C03648=1141.672,169.284,-60.274,-178.490,7.173,148.902
C03649=1141.677,169.034,-60.251,-178.493,7.171,148.902
C03650=1141.681,168.786,-60.228,-178.496,7.169,148.903
C03651=1141.685,168.537,-60.206,-178.499,7.167,148.903
C03652=1141.690,168.288,-60.185,-178.501,7.165,148.903
C03653=1141.695,168.039,-60.162,-178.505,7.162,148.903
C03654=1141.699,167.790,-60.139,-178.507,7.160,148.904
C03655=1141.704,167.541,-60.118,-178.510,7.158,148.904
C03656=1141.708,167.292,-60.096,-178.513,7.156,148.904
C03657=1141.714,167.043,-60.073,-178.516,7.154,148.905
C03658=1141.718,166.794,-60.051,-178.518,7.151,148.905
C03659=1141.723,166.546,-60.029,-178.521,7.150,148.905
C03660=1141.727,166.296,-60.007,-178.524,7.147,148.906
C03661=1141.733,166.047,-59.985,-178.527,7.145,148.906
C03662=1141.737,165.798,-59.963,-178.529,7.143,148.906
C03663=1141.742,165.549,-59.941,-178.533,7.141,148.906
C03664=1141.746,165.300,-59.919,-178.535,7.139,148.907
C03665=1141.751,165.051,-59.897,-178.538,7.137,148.907
C03666=1141.755,164.802,-59.875,-178.541,7.134,148.907
C03667=1141.761,164.553,-59.853,-178.544,7.133,148.908
C03668=1141.765,164.304,-59.830,-178.547,7.130,148.908
C03669=1141.770,164.056,-59.808,-178.549,7.128,148.908
C03670=1141.774,163.806,-59.786,-178.552,7.126,148.909
C03671=1141.779,163.558,-59.765,-178.555,7.124,148.909
C03672=1141.783,163.308,-59.743,-178.558,7.122,148.909
C03673=1141.788,163.060,-59.721,-178.560,7.120,148.909
C03674=1141.792,162.811,-59.699,-178.563,7.118,148.910
C03675=1141.798,162.562,-59.677,-178.566,7.116,148.910
C03676=1141.803,162.313,-59.655,-178.569,7.113,148.911
C03677=1141.807,162.063,-59.634,-178.572,7.111,148.911
C03678=1141.812,161.814,-59.612,-178.574,7.110,148.911
C03679=1141.816,161.565,-59.590,-178.578,7.107,148.911
C03680=1141.821,161.316,-59.568,-178.580,7.105,148.912
C03681=1141.826,161.067,-59.546,-178.583,7.103,148.912
C03682=1141.830,160.818,-59.524,-178.586,7.101,148.912
C03683=1141.835,160.570,-59.503,-178.589,7.099,148.913
C03684=1141.840,160.320,-59.481,-178.591,7.097,148.913
C03685=1141.844,160.072,-59.459,-178.594,7.094,148.913
C03686=1141.849,159.822,-59.438,-178.597,7.093,148.914
C03687=1141.854,159.573,-59.416,-178.599,7.091,148.914
C03688=1141.859,159.324,-59.394,-178.603,7.088,148.914
C03689=1141.863,159.075,-59.372,-178.605,7.087,148.915
C03690=1141.868,158.827,-59.351,-178.608,7.085,148.915
C03691=1141.873,158.578,-59.329,-178.611,7.082,148.915
C03692=1141.877,158.328,-59.308,-178.614,7.080,148.916
C03693=1141.882,158.079,-59.286,-178.616,7.079,148.916
C03694=1141.887,157.810,-59.263,-178.620,7.076,148.916
C03695=1141.892,157.541,-59.239,-178.623,7.074,148.917
C03696=1141.897,157.272,-59.216,-178.625,7.072,148.917
C03697=1141.902,157.003,-59.193,-178.629,7.069,148.917
C03698=1141.907,156.754,-59.171,-178.631,7.067,148.918
C03699=1141.911,156.505,-59.149,-178.634,7.066,148.918
C03700=1141.916,156.256,-59.129,-178.637,7.063,148.918
C03701=1141.921,156.008,-59.107,-178.640,7.061,148.919
C03702=1141.925,155.758,-59.085,-178.642,7.059,148.919
C03703=1141.930,155.509,-59.064,-178.646,7.057,148.919
C03704=1141.935,155.260,-59.042,-178.648,7.055,148.920
C03705=1141.940,155.012,-59.021,-178.651,7.053,148.920
C03706=1141.945,154.762,-58.999,-178.654,7.051,148.920
C03707=1141.949,154.513,-58.978,-178.656,7.049,148.921
C03708=1141.954,154.264,-58.957,-178.659,7.047,148.921
C03709=1141.959,154.015,-58.936,-178.662,7.045,148.921
C03710=1141.963,153.765,-58.914,-178.665,7.043,148.922
C03711=1141.968,153.517,-58.893,-178.668,7.041,148.922
C03712=1141.973,153.268,-58.872,-178.671,7.039,148.922
C03713=1141.977,153.019,-58.851,-178.673,7.036,148.923
C03714=1141.982,152.769,-58.829,-178.676,7.035,148.923
C03715=1141.987,152.521,-58.808,-178.679,7.033,148.923
C03716=1141.992,152.271,-58.787,-178.682,7.031,148.924
C03717=1141.996,152.023,-58.766,-178.685,7.029,148.924
C03718=1142.001,151.773,-58.744,-178.688,7.027,148.925
C03719=1142.006,151.524,-58.722,-178.690,7.025,148.925
C03720=1142.011,151.275,-58.702,-178.693,7.022,148.925
C03721=1142.015,151.027,-58.680,-178.696,7.021,148.925
C03722=1142.020,150.778,-58.659,-178.699,7.019,148.926
C03723=1142.025,150.528,-58.638,-178.701,7.017,148.926
C03724=1142.029,150.279,-58.617,-178.705,7.015,148.927
C03725=1142.034,150.030,-58.596,-178.707,7.013,148.927
C03726=1142.039,149.781,-58.574,-178.709,7.011,148.927
C03727=1142.043,149.532,-58.554,-178.712,7.009,148.927
C03728=1142.048,149.282,-58.533,-178.716,7.007,148.928
C03729=1142.053,149.034,-58.511,-178.718,7.005,148.928
C03730=1142.057,148.785,-58.491,-178.721,7.003,148.929
C03731=1142.062,148.536,-58.470,-178.724,7.002,148.929
C03732=1142.068,148.286,-58.449,-178.727,6.999,148.929
C03733=1142.072,148.038,-58.428,-178.729,6.997,148.930
C03734=1142.077,147.789,-58.407,-178.732,6.995,148.930
C03735=1142.081,147.539,-58.385,-178.735,6.994,148.930
C03736=1142.086,147.290,-58.365,-178.738,6.991,148.931
C03737=1142.091,147.041,-58.343,-178.741,6.989,148.931
C03738=1142.095,146.792,-58.323,-178.743,6.988,148.931
C03739=1142.100,146.543,-58.302,-178.746,6.986,148.932
C03740=1142.105,146.294,-58.282,-178.749,6.983,148.932
C03741=1142.110,146.045,-58.261,-178.752,6.981,148.932
C03742=1142.115,145.796,-58.239,-178.754,6.980,148.933
C03743=1142.119,145.547,-58.219,-178.757,6.978,148.933
C03744=1142.124,145.297,-58.197,-178.760,6.975,148.934
C03745=1142.128,145.048,-58.177,-178.763,6.974,148.934
C03746=1142.133,144.799,-58.156,-178.766,6.972,148.934
C03747=1142.138,144.550,-58.135,-178.768,6.970,148.935
C03748=1142.143,144.301,-58.115,-178.771,6.969,148.935
C03749=1142.147,144.053,-58.093,-178.774,6.966,148.935
C03750=1142.152,143.803,-58.072,-178.777,6.964,148.936
C03751=1142.157,143.554,-58.052,-178.779,6.962,148.936
C03752=1142.162,143.305,-58.031,-178.782,6.961,148.936
C03753=1142.166,143.056,-58.011,-178.785,6.958,148.937
C03754=1142.172,142.807,-57.990,-178.788,6.956,148.937
C03755=1142.176,142.558,-57.969,-178.791,6.955,148.938
C03756=1142.180,142.309,-57.949,-178.794,6.953,148.938
C03757=1142.186,142.060,-57.928,-178.796,6.951,148.938
C03758=1142.190,141.811,-57.908,-178.800,6.949,148.939
C03759=1142.195,141.562,-57.887,-178.802,6.947,148.939
C03760=1142.200,141.313,-57.866,-178.805,6.945,148.939
C03761=1142.204,141.064,-57.846,-178.807,6.943,148.940
C03762=1142.209,140.814,-57.825,-178.810,6.942,148.940
C03763=1142.214,140.565,-57.805,-178.813,6.939,148.940
C03764=1142.219,140.316,-57.784,-178.816,6.937,148.941
C03765=1142.224,140.067,-57.764,-178.819,6.936,148.941
C03766=1142.228,139.818,-57.744,-178.821,6.934,148.942
C03767=1142.233,139.568,-57.723,-178.824,6.932,148.942
C03768=1142.238,139.319,-57.702,-178.827,6.931,148.942
C03769=1142.242,139.070,-57.682,-178.830,6.928,148.943
C03770=1142.247,138.821,-57.661,-178.833,6.926,148.943
C03771=1142.252,138.572,-57.641,-178.836,6.925,148.944
C03772=1142.256,138.323,-57.621,-178.838,6.923,148.944
C03773=1142.262,138.073,-57.600,-178.841,6.921,148.944
C03774=1142.266,137.824,-57.580,-178.843,6.919,148.944
C03775=1142.271,137.576,-57.559,-178.847,6.917,148.945
C03776=1142.275,137.327,-57.539,-178.849,6.915,148.945
C03777=1142.280,137.077,-57.519,-178.852,6.913,148.946
C03778=1142.285,136.828,-57.498,-178.855,6.912,148.946
C03779=1142.289,136.579,-57.478,-178.857,6.910,148.946
C03780=1142.294,136.330,-57.457,-178.860,6.908,148.947
C03781=1142.300,136.081,-57.438,-178.864,6.906,148.947
C03782=1142.304,135.832,-57.417,-178.866,6.904,148.948
C03783=1142.309,135.583,-57.397,-178.869,6.902,148.948
C03784=1142.313,135.333,-57.377,-178.872,6.901,148.948
C03785=1142.319,135.084,-57.356,-178.874,6.899,148.949
C03786=1142.323,134.835,-57.336,-178.877,6.897,148.949
C03787=1142.328,134.585,-57.316,-178.880,6.895,148.950
C03788=1142.332,134.336,-57.296,-178.883,6.893,148.950
C03789=1142.337,134.088,-57.275,-178.886,6.891,148.950
C03790=1142.343,133.838,-57.256,-178.889,6.890,148.951
C03791=1142.347,133.589,-57.235,-178.891,6.888,148.951
C03792=1142.352,133.340,-57.215,-178.894,6.886,148.951
C03793=1142.356,133.091,-57.195,-178.897,6.884,148.952
C03794=1142.361,132.842,-57.175,-178.899,6.883,148.952
C03795=1142.366,132.592,-57.155,-178.903,6.880,148.953
C03796=1142.371,132.344,-57.135,-178.905,6.878,148.953
C03797=1142.376,132.094,-57.115,-178.908,6.876,148.953
C03798=1142.381,131.826,-57.093,-178.911,6.875,148.954
C03799=1142.386,131.557,-57.071,-178.914,6.873,148.954
C03800=1142.391,131.289,-57.050,-178.917,6.871,148.955
C03801=1142.396,131.021,-57.029,-178.920,6.869,148.955
C03802=1142.401,130.771,-57.008,-178.922,6.867,148.955
C03803=1142.406,130.522,-56.988,-178.926,6.865,148.956
C03804=1142.411,130.273,-56.969,-178.928,6.863,148.956
C03805=1142.416,130.023,-56.949,-178.931,6.862,148.957
C03806=1142.420,129.774,-56.929,-178.934,6.860,148.957
C03807=1142.425,129.525,-56.909,-178.937,6.858,148.957
C03808=1142.429,129.276,-56.889,-178.939,6.856,148.958
C03809=1142.435,129.027,-56.869,-178.942,6.855,148.958
C03810=1142.439,128.778,-56.849,-178.945,6.853,148.959
C03811=1142.444,128.528,-56.829,-178.947,6.851,148.959
C03812=1142.449,128.279,-56.810,-178.950,6.850,148.959
C03813=1142.454,128.031,-56.790,-178.953,6.847,148.960
C03814=1142.459,127.781,-56.770,-178.956,6.845,148.960
C03815=1142.463,127.532,-56.750,-178.959,6.844,148.961
C03816=1142.468,127.283,-56.730,-178.962,6.842,148.961
C03817=1142.473,127.034,-56.711,-178.964,6.840,148.961
C03818=1142.478,126.784,-56.691,-178.967,6.839,148.962
C03819=1142.483,126.535,-56.671,-178.970,6.837,148.962
C03820=1142.488,126.286,-56.651,-178.973,6.835,148.963
C03821=1142.492,126.037,-56.632,-178.975,6.834,148.963
C03822=1142.497,125.787,-56.612,-178.978,6.832,148.963
C03823=1142.501,125.539,-56.592,-178.981,6.830,148.964
C03824=1142.506,125.290,-56.573,-178.983,6.829,148.964
C03825=1142.511,125.040,-56.553,-178.986,6.827,148.965
C03826=1142.516,124.791,-56.534,-178.989,6.824,148.965
C03827=1142.521,124.542,-56.514,-178.992,6.823,148.965
C03828=1142.525,124.293,-56.494,-178.995,6.821,148.966
C03829=1142.530,124.043,-56.474,-178.998,6.819,148.966
C03830=1142.535,123.794,-56.455,-179.000,6.818,148.967
C03831=1142.539,123.545,-56.436,-179.003,6.816,148.967
C03832=1142.544,123.295,-56.416,-179.006,6.814,148.967
C03833=1142.550,123.047,-56.397,-179.009,6.812,148.968
C03834=1142.554,122.797,-56.377,-179.011,6.811,148.968
C03835=1142.559,122.549,-56.357,-179.014,6.809,148.969
C03836=1142.564,122.299,-56.338,-179.017,6.807,148.969
C03837=1142.568,122.050,-56.319,-179.020,6.806,148.970
C03838=1142.573,121.801,-56.299,-179.023,6.804,148.970
C03839=1142.578,121.552,-56.280,-179.025,6.803,148.970
C03840=1142.583,121.302,-56.260,-179.028,6.801,148.971
C03841=1142.588,121.053,-56.241,-179.031,6.799,148.971
C03842=1142.592,120.804,-56.222,-179.034,6.798,148.972
C03843=1142.598,120.555,-56.202,-179.036,6.796,148.972
C03844=1142.602,120.305,-56.183,-179.039,6.794,148.972
C03845=1142.607,120.056,-56.163,-179.042,6.792,148.973
C03846=1142.612,119.807,-56.144,-179.045,6.790,148.973
C03847=1142.616,119.558,-56.125,-179.048,6.788,148.974
C03848=1142.622,119.309,-56.105,-179.050,6.787,148.974
C03849=1142.627,119.059,-56.086,-179.053,6.785,148.974
C03850=1142.631,118.811,-56.067,-179.056,6.783,148.975
C03851=1142.636,118.561,-56.047,-179.059,6.782,148.975
C03852=1142.641,118.312,-56.028,-179.061,6.780,148.976
C03853=1142.645,118.063,-56.009,-179.064,6.778,148.976
C03854=1142.650,117.813,-55.990,-179.067,6.776,148.976
C03855=1142.656,117.564,-55.971,-179.070,6.775,148.977
C03856=1142.660,117.315,-55.952,-179.073,6.773,148.977
C03857=1142.665,117.066,-55.932,-179.075,6.772,148.978
C03858=1142.670,116.816,-55.913,-179.078,6.770,148.978
C03859=1142.674,116.568,-55.894,-179.081,6.768,148.979
C03860=1142.679,116.318,-55.874,-179.084,6.767,148.979
C03861=1142.685,116.069,-55.856,-179.086,6.765,148.979
C03862=1142.689,115.819,-55.837,-179.089,6.763,148.980
C03863=1142.694,115.571,-55.818,-179.092,6.762,148.980
C03864=1142.699,115.321,-55.798,-179.095,6.760,148.981
C03865=1142.703,115.072,-55.779,-179.097,6.758,148.981
C03866=1142.708,114.822,-55.760,-179.100,6.757,148.981
C03867=1142.713,114.574,-55.742,-179.103,6.755,148.982
C03868=1142.718,114.324,-55.722,-179.106,6.754,148.983
C03869=1142.723,114.075,-55.704,-179.109,6.752,148.983
C03870=1142.727,113.825,-55.684,-179.111,6.750,148.983
C03871=1142.733,113.576,-55.665,-179.114,6.748,148.984
C03872=1142.737,113.328,-55.646,-179.117,6.747,148.984
C03873=1142.742,113.078,-55.627,-179.120,6.745,148.985
C03874=1142.747,112.829,-55.609,-179.122,6.743,148.985
C03875=1142.752,112.580,-55.589,-179.125,6.742,148.985
C03876=1142.757,112.330,-55.571,-179.127,6.741,148.986
C03877=1142.761,112.081,-55.551,-179.130,6.739,148.986
C03878=1142.766,111.832,-55.533,-179.133,6.738,148.987
C03879=1142.772,111.583,-55.514,-179.136,6.736,148.987
C03880=1142.776,111.334,-55.495,-179.139,6.734,148.988
C03881=1142.781,111.084,-55.476,-179.141,6.733,148.988
C03882=1142.785,110.835,-55.457,-179.144,6.731,148.988
C03883=1142.791,110.585,-55.439,-179.147,6.729,148.989
C03884=1142.796,110.337,-55.420,-179.149,6.728,148.989
C03885=1142.800,110.087,-55.400,-179.152,6.726,148.990
C03886=1142.805,109.838,-55.382,-179.155,6.724,148.990
C03887=1142.810,109.588,-55.363,-179.158,6.723,148.991
C03888=1142.815,109.339,-55.345,-179.161,6.721,148.991
C03889=1142.820,109.091,-55.326,-179.164,6.720,148.992
C03890=1142.825,108.841,-55.307,-179.166,6.718,148.992
C03891=1142.829,108.592,-55.289,-179.169,6.716,148.992
C03892=1142.835,108.342,-55.270,-179.172,6.715,148.993
C03893=1142.839,108.093,-55.251,-179.175,6.713,148.993
C03894=1142.844,107.844,-55.233,-179.177,6.711,148.994
C03895=1142.849,107.595,-55.214,-179.180,6.710,148.994
C03896=1142.853,107.345,-55.195,-179.183,6.708,148.995
C03897=1142.858,107.096,-55.177,-179.185,6.707,148.995
C03898=1142.864,106.847,-55.158,-179.188,6.706,148.995
C03899=1142.868,106.597,-55.140,-179.191,6.704,148.996
C03900=1142.873,106.349,-55.121,-179.194,6.702,148.996
C03901=1142.878,106.099,-55.102,-179.196,6.701,148.997
C03902=1142.883,105.830,-55.083,-179.199,6.699,148.997
C03903=1142.888,105.562,-55.062,-179.202,6.698,148.998
C03904=1142.893,105.294,-55.042,-179.206,6.695,148.998
C03905=1142.899,105.026,-55.022,-179.208,6.693,148.999
C03906=1142.903,104.776,-55.004,-179.211,6.692,148.999
C03907=1142.908,104.527,-54.985,-179.214,6.690,149.000
C03908=1142.914,104.278,-54.967,-179.216,6.690,149.000
C03909=1142.919,104.029,-54.949,-179.219,6.688,149.000
C03910=1142.923,103.779,-54.931,-179.222,6.686,149.001
C03911=1142.928,103.530,-54.912,-179.225,6.684,149.001
C03912=1142.933,103.281,-54.893,-179.227,6.683,149.002
C03913=1142.938,103.031,-54.875,-179.230,6.681,149.002
C03914=1142.942,102.782,-54.857,-179.233,6.680,149.003
C03915=1142.947,102.533,-54.838,-179.236,6.678,149.003
C03916=1142.952,102.284,-54.820,-179.239,6.676,149.004
C03917=1142.958,102.034,-54.802,-179.241,6.675,149.004
C03918=1142.962,101.784,-54.783,-179.244,6.674,149.004
C03919=1142.967,101.536,-54.765,-179.247,6.673,149.005
C03920=1142.971,101.287,-54.747,-179.249,6.671,149.005
C03921=1142.976,101.038,-54.729,-179.252,6.669,149.006
C03922=1142.982,100.788,-54.710,-179.255,6.668,149.006
C03923=1142.986,100.538,-54.692,-179.258,6.666,149.007
C03924=1142.991,100.289,-54.674,-179.260,6.664,149.007
C03925=1142.996,100.040,-54.656,-179.264,6.663,149.008
C03926=1143.001,99.791,-54.638,-179.266,6.661,149.008
C03927=1143.006,99.542,-54.619,-179.268,6.660,149.009
C03928=1143.011,99.292,-54.600,-179.271,6.659,149.009
C03929=1143.016,99.043,-54.582,-179.274,6.657,149.009
C03930=1143.021,98.794,-54.564,-179.277,6.655,149.010
C03931=1143.025,98.544,-54.546,-179.280,6.654,149.010
C03932=1143.030,98.295,-54.528,-179.283,6.652,149.011
C03933=1143.035,98.046,-54.510,-179.285,6.651,149.011
C03934=1143.040,97.796,-54.492,-179.288,6.650,149.012
C03935=1143.044,97.547,-54.474,-179.290,6.648,149.012
C03936=1143.049,97.298,-54.456,-179.293,6.646,149.013
C03937=1143.054,97.049,-54.438,-179.296,6.645,149.013
C03938=1143.059,96.799,-54.420,-179.299,6.643,149.014
C03939=1143.064,96.550,-54.402,-179.302,6.642,149.014
C03940=1143.070,96.301,-54.383,-179.304,6.640,149.014
C03941=1143.074,96.051,-54.365,-179.307,6.639,149.015
C03942=1143.079,95.802,-54.347,-179.310,6.638,149.015
C03943=1143.084,95.553,-54.329,-179.312,6.636,149.016
C03944=1143.089,95.303,-54.311,-179.315,6.635,149.016
C03945=1143.094,95.054,-54.294,-179.318,6.633,149.017
C03946=1143.099,94.804,-54.276,-179.321,6.631,149.017
C03947=1143.104,94.555,-54.258,-179.323,6.629,149.018
C03948=1143.109,94.306,-54.240,-179.326,6.629,149.018
C03949=1143.114,94.057,-54.222,-179.329,6.627,149.019
C03950=1143.119,93.808,-54.204,-179.332,6.626,149.019
C03951=1143.124,93.559,-54.186,-179.334,6.624,149.019
C03952=1143.128,93.309,-54.169,-179.337,6.622,149.020
C03953=1143.132,93.059,-54.151,-179.340,6.622,149.021
C03954=1143.137,92.810,-54.133,-179.342,6.620,149.021
C03955=1143.142,92.561,-54.115,-179.345,6.618,149.021
C03956=1143.147,92.312,-54.097,-179.348,6.617,149.022
C03957=1143.152,92.062,-54.080,-179.351,6.615,149.022
C03958=1143.157,91.813,-54.062,-179.354,6.614,149.023
C03959=1143.162,91.564,-54.044,-179.356,6.613,149.023
C03960=1143.167,91.314,-54.026,-179.359,6.611,149.024
C03961=1143.172,91.065,-54.009,-179.361,6.610,149.024
C03962=1143.177,90.815,-53.991,-179.364,6.608,149.025
C03963=1143.181,90.567,-53.973,-179.367,6.607,149.025
C03964=1143.186,90.317,-53.955,-179.370,6.606,149.026
C03965=1143.191,90.068,-53.938,-179.372,6.604,149.026
C03966=1143.196,89.818,-53.920,-179.375,6.602,149.026
C03967=1143.201,89.569,-53.902,-179.378,6.601,149.027
C03968=1143.206,89.319,-53.885,-179.381,6.599,149.028
C03969=1143.211,89.070,-53.867,-179.383,6.599,149.028
C03970=1143.216,88.821,-53.849,-179.386,6.597,149.028
C03971=1143.221,88.572,-53.832,-179.389,6.595,149.029
C03972=1143.226,88.322,-53.814,-179.392,6.594,149.029
C03973=1143.231,88.073,-53.797,-179.395,6.592,149.030
C03974=1143.236,87.823,-53.779,-179.397,6.591,149.030
C03975=1143.240,87.575,-53.762,-179.399,6.590,149.031
C03976=1143.245,87.325,-53.744,-179.403,6.588,149.031
C03977=1143.250,87.076,-53.726,-179.405,6.587,149.032
C03978=1143.255,86.826,-53.709,-179.408,6.585,149.032
C03979=1143.260,86.578,-53.692,-179.410,6.584,149.033
C03980=1143.265,86.328,-53.675,-179.413,6.582,149.033
C03981=1143.270,86.079,-53.657,-179.416,6.581,149.034
C03982=1143.275,85.829,-53.639,-179.419,6.580,149.034
C03983=1143.280,85.580,-53.622,-179.421,6.579,149.035
C03984=1143.285,85.330,-53.605,-179.424,6.577,149.035
C03985=1143.290,85.081,-53.587,-179.427,6.576,149.036
C03986=1143.295,84.831,-53.570,-179.430,6.574,149.036
C03987=1143.299,84.582,-53.552,-179.432,6.573,149.036
C03988=1143.304,84.333,-53.535,-179.435,6.571,149.037
C03989=1143.309,84.083,-53.517,-179.438,6.570,149.038
C03990=1143.314,83.834,-53.500,-179.441,6.569,149.038
C03991=1143.319,83.585,-53.483,-179.443,6.568,149.038
C03992=1143.324,83.336,-53.465,-179.446,6.566,149.039
C03993=1143.329,83.086,-53.449,-179.449,6.565,149.039
C03994=1143.334,82.837,-53.431,-179.451,6.563,149.040
C03995=1143.339,82.587,-53.414,-179.454,6.562,149.040
C03996=1143.343,82.338,-53.396,-179.456,6.560,149.041
C03997=1143.348,82.089,-53.379,-179.460,6.559,149.041
C03998=1143.354,81.839,-53.362,-179.462,6.558,149.042
C03999=1143.358,81.591,-53.345,-179.464,6.557,149.042
C04000=1143.364,81.341,-53.327,-179.467,6.555,149.043
C04001=1143.368,81.091,-53.311,-179.470,6.554,149.043
C04002=1143.373,80.842,-53.293,-179.473,6.552,149.044
C04003=1143.378,80.592,-53.275,-179.475,6.551,149.044
C04004=1143.383,80.344,-53.259,-179.478,6.549,149.045
C04005=1143.389,80.094,-53.242,-179.481,6.548,149.045
C04006=1143.393,79.826,-53.223,-179.484,6.547,149.046
C04007=1143.398,79.557,-53.204,-179.487,6.545,149.046
C04008=1143.404,79.289,-53.186,-179.490,6.544,149.047
C04009=1143.409,79.020,-53.168,-179.493,6.542,149.047
C04010=1143.414,78.770,-53.151,-179.495,6.541,149.048
C04011=1143.419,78.522,-53.134,-179.498,6.540,149.048
C04012=1143.424,78.272,-53.116,-179.501,6.538,149.049
C04013=1143.429,78.023,-53.100,-179.503,6.537,149.049
C04014=1143.434,77.773,-53.082,-179.506,6.536,149.050
C04015=1143.439,77.524,-53.066,-179.509,6.534,149.050
C04016=1143.444,77.275,-53.049,-179.512,6.533,149.051
C04017=1143.449,77.025,-53.032,-179.514,6.532,149.051
C04018=1143.454,76.776,-53.014,-179.517,6.530,149.052
C04019=1143.459,76.527,-52.998,-179.520,6.529,149.052
C04020=1143.464,76.277,-52.981,-179.522,6.528,149.053
C04021=1143.468,76.028,-52.964,-179.525,6.526,149.053
C04022=1143.474,75.778,-52.947,-179.528,6.525,149.054
C04023=1143.479,75.529,-52.930,-179.530,6.524,149.054
C04024=1143.484,75.279,-52.913,-179.533,6.522,149.055
C04025=1143.488,75.030,-52.896,-179.536,6.521,149.055
C04026=1143.493,74.781,-52.880,-179.539,6.520,149.056
C04027=1143.499,74.531,-52.863,-179.541,6.519,149.056
C04028=1143.503,74.282,-52.846,-179.544,6.517,149.056
C04029=1143.508,74.032,-52.829,-179.547,6.516,149.057
C04030=1143.513,73.783,-52.813,-179.549,6.515,149.058
C04031=1143.518,73.534,-52.796,-179.552,6.513,149.058
C04032=1143.523,73.284,-52.779,-179.555,6.512,149.059
C04033=1143.528,73.035,-52.762,-179.557,6.511,149.059
C04034=1143.533,72.785,-52.745,-179.560,6.509,149.060
C04035=1143.538,72.536,-52.728,-179.563,6.508,149.060
C04036=1143.543,72.287,-52.712,-179.565,6.507,149.061
C04037=1143.548,72.037,-52.695,-179.568,6.506,149.061
C04038=1143.553,71.788,-52.678,-179.571,6.504,149.061
C04039=1143.558,71.539,-52.662,-179.573,6.503,149.062
C04040=1143.563,71.289,-52.645,-179.576,6.502,149.063
C04041=1143.567,71.040,-52.628,-179.579,6.500,149.063
C04042=1143.573,70.791,-52.612,-179.581,6.499,149.063
C04043=1143.577,70.542,-52.595,-179.584,6.498,149.064
C04044=1143.582,70.292,-52.578,-179.587,6.496,149.065
C04045=1143.588,70.042,-52.562,-179.589,6.495,149.065
C04046=1143.592,69.793,-52.546,-179.592,6.494,149.066
C04047=1143.597,69.543,-52.528,-179.595,6.492,149.066
C04048=1143.602,69.294,-52.512,-179.597,6.492,149.066
C04049=1143.607,69.045,-52.495,-179.600,6.490,149.067
C04050=1143.612,68.796,-52.479,-179.603,6.489,149.068
C04051=1143.618,68.546,-52.462,-179.605,6.488,149.068
C04052=1143.622,68.296,-52.446,-179.608,6.486,149.068
C04053=1143.627,68.047,-52.429,-179.611,6.485,149.069
C04054=1143.632,67.798,-52.413,-179.614,6.484,149.070
C04055=1143.637,67.549,-52.396,-179.616,6.482,149.070
C04056=1143.642,67.299,-52.380,-179.619,6.482,149.071
C04057=1143.647,67.049,-52.363,-179.622,6.480,149.071
C04058=1143.652,66.800,-52.347,-179.624,6.479,149.071
C04059=1143.656,66.551,-52.330,-179.627,6.478,149.072
C04060=1143.662,66.301,-52.314,-179.630,6.476,149.073
C04061=1143.667,66.052,-52.297,-179.633,6.475,149.073
C04062=1143.672,65.803,-52.281,-179.635,6.474,149.073
C04063=1143.677,65.553,-52.265,-179.638,6.473,149.074
C04064=1143.682,65.304,-52.249,-179.640,6.472,149.075
C04065=1143.686,65.055,-52.232,-179.643,6.470,149.075
C04066=1143.691,64.805,-52.216,-179.646,6.469,149.076
C04067=1143.697,64.555,-52.199,-179.648,6.468,149.076
C04068=1143.701,64.306,-52.183,-179.651,6.466,149.077
C04069=1143.707,64.057,-52.167,-179.654,6.465,149.077
C04070=1143.711,63.807,-52.150,-179.656,6.464,149.078
C04071=1143.716,63.558,-52.134,-179.659,6.463,149.078
C04072=1143.721,63.308,-52.118,-179.662,6.462,149.079
C04073=1143.726,63.059,-52.102,-179.665,6.460,149.079
C04074=1143.731,62.809,-52.086,-179.667,6.459,149.080
C04075=1143.736,62.561,-52.070,-179.670,6.458,149.080
C04076=1143.742,62.310,-52.053,-179.673,6.457,149.081
C04077=1143.747,62.061,-52.037,-179.675,6.456,149.081
C04078=1143.751,61.811,-52.021,-179.678,6.454,149.082
C04079=1143.756,61.562,-52.005,-179.681,6.453,149.082
C04080=1143.761,61.313,-51.988,-179.683,6.452,149.083
C04081=1143.766,61.064,-51.972,-179.686,6.450,149.083
C04082=1143.771,60.814,-51.956,-179.688,6.450,149.084
C04083=1143.776,60.565,-51.940,-179.691,6.448,149.084
C04084=1143.782,60.315,-51.924,-179.694,6.447,149.085
C04085=1143.786,60.066,-51.908,-179.696,6.446,149.085
C04086=1143.791,59.816,-51.892,-179.699,6.444,149.086
C04087=1143.796,59.567,-51.875,-179.701,6.444,149.086
C04088=1143.801,59.317,-51.860,-179.705,6.442,149.087
C04089=1143.806,59.068,-51.843,-179.707,6.441,149.087
C04090=1143.811,58.819,-51.828,-179.710,6.440,149.088
C04091=1143.816,58.569,-51.811,-179.713,6.439,149.088
C04092=1143.821,58.320,-51.795,-179.715,6.438,149.089
C04093=1143.826,58.070,-51.780,-179.718,6.436,149.089
C04094=1143.831,57.821,-51.763,-179.720,6.436,149.090
C04095=1143.836,57.571,-51.748,-179.723,6.434,149.090
C04096=1143.841,57.321,-51.732,-179.725,6.433,149.091
C04097=1143.846,57.073,-51.715,-179.728,6.432,149.091
C04098=1143.851,56.823,-51.700,-179.731,6.430,149.092
C04099=1143.856,56.573,-51.684,-179.733,6.429,149.092
C04100=1143.861,56.325,-51.668,-179.737,6.428,149.093
C04101=1143.866,56.075,-51.652,-179.739,6.427,149.093
C04102=1143.871,55.825,-51.636,-179.742,6.426,149.094
C04103=1143.876,55.576,-51.620,-179.744,6.425,149.095
C04104=1143.881,55.326,-51.604,-179.747,6.423,149.095
C04105=1143.886,55.077,-51.589,-179.749,6.423,149.095
C04106=1143.891,54.827,-51.573,-179.752,6.421,149.096
C04107=1143.896,54.578,-51.556,-179.754,6.420,149.097
C04108=1143.901,54.329,-51.541,-179.757,6.419,149.097
C04109=1143.906,54.079,-51.526,-179.760,6.418,149.098
C04110=1143.912,53.811,-51.509,-179.763,6.417,149.098
C04111=1143.917,53.542,-51.491,-179.766,6.415,149.099
C04112=1143.922,53.273,-51.474,-179.769,6.414,149.099
C04113=1143.928,53.005,-51.457,-179.771,6.413,149.100
C04114=1143.933,52.755,-51.442,-179.774,6.412,149.100
C04115=1143.937,52.506,-51.426,-179.777,6.410,149.101
C04116=1143.942,52.256,-51.411,-179.779,6.410,149.101
C04117=1143.948,52.007,-51.395,-179.782,6.408,149.102
C04118=1143.953,51.758,-51.379,-179.785,6.407,149.103
C04119=1143.958,51.508,-51.363,-179.788,6.406,149.103
C04120=1143.962,51.259,-51.348,-179.790,6.405,149.103
C04121=1143.968,51.009,-51.332,-179.793,6.404,149.104
C04122=1143.973,50.759,-51.316,-179.795,6.403,149.105
C04123=1143.978,50.510,-51.301,-179.798,6.401,149.105
C04124=1143.983,50.261,-51.286,-179.800,6.401,149.106
C04125=1143.988,50.011,-51.270,-179.803,6.399,149.106
C04126=1143.992,49.762,-51.254,-179.806,6.399,149.107
C04127=1143.998,49.512,-51.238,-179.809,6.397,149.107
C04128=1144.002,49.263,-51.223,-179.811,6.396,149.108
C04129=1144.007,49.013,-51.207,-179.814,6.395,149.108
C04130=1144.013,48.764,-51.191,-179.816,6.394,149.109
C04131=1144.017,48.515,-51.177,-179.819,6.392,149.109
C04132=1144.023,48.265,-51.161,-179.822,6.392,149.110
C04133=1144.027,48.015,-51.145,-179.824,6.390,149.110
C04134=1144.032,47.766,-51.130,-179.826,6.389,149.111
C04135=1144.038,47.517,-51.114,-179.830,6.388,149.111
C04136=1144.043,47.267,-51.099,-179.832,6.387,149.112
C04137=1144.048,47.018,-51.084,-179.835,6.386,149.113
C04138=1144.052,46.768,-51.068,-179.837,6.385,149.113
C04139=1144.058,46.519,-51.052,-179.840,6.384,149.113
C04140=1144.063,46.269,-51.038,-179.843,6.383,149.114
C04141=1144.068,46.020,-51.022,-179.845,6.381,149.115
C04142=1144.073,45.770,-51.007,-179.848,6.381,149.115
C04143=1144.077,45.520,-50.991,-179.851,6.379,149.116
C04144=1144.083,45.271,-50.976,-179.853,6.379,149.116
C04145=1144.088,45.022,-50.960,-179.856,6.377,149.117
C04146=1144.093,44.773,-50.945,-179.858,6.376,149.117
C04147=1144.098,44.523,-50.930,-179.861,6.375,149.118
C04148=1144.103,44.274,-50.915,-179.864,6.374,149.118
C04149=1144.108,44.023,-50.899,-179.867,6.373,149.119
C04150=1144.113,43.774,-50.884,-179.869,6.372,149.119
C04151=1144.118,43.525,-50.869,-179.871,6.371,149.120
C04152=1144.123,43.275,-50.853,-179.874,6.370,149.120
C04153=1144.128,43.026,-50.838,-179.876,6.369,149.121
C04154=1144.134,42.777,-50.823,-179.879,6.368,149.121
C04155=1144.138,42.527,-50.808,-179.882,6.367,149.122
C04156=1144.143,42.277,-50.792,-179.885,6.366,149.123
C04157=1144.148,42.028,-50.777,-179.887,6.365,149.123
C04158=1144.153,41.779,-50.762,-179.890,6.363,149.124
C04159=1144.158,41.529,-50.748,-179.892,6.363,149.124
C04160=1144.164,41.280,-50.732,-179.895,6.361,149.125
C04161=1144.168,41.030,-50.717,-179.897,6.360,149.125
C04162=1144.174,40.781,-50.701,-179.900,6.360,149.126
C04163=1144.179,40.531,-50.687,-179.903,6.358,149.126
C04164=1144.183,40.281,-50.671,-179.905,6.358,149.127
C04165=1144.188,40.032,-50.656,-179.908,6.356,149.127
C04166=1144.194,39.782,-50.641,-179.910,6.355,149.128
C04167=1144.198,39.533,-50.626,-179.914,6.354,149.128
C04168=1144.204,39.284,-50.611,-179.916,6.353,149.129
C04169=1144.209,39.034,-50.597,-179.919,6.351,149.129
C04170=1144.214,38.785,-50.581,-179.921,6.351,149.130
C04171=1144.219,38.535,-50.566,-179.923,6.350,149.130
C04172=1144.224,38.286,-50.552,-179.927,6.349,149.131
C04173=1144.229,38.036,-50.536,-179.929,6.348,149.132
C04174=1144.234,37.787,-50.522,-179.931,6.346,149.132
C04175=1144.239,37.537,-50.506,-179.934,6.346,149.133
C04176=1144.244,37.288,-50.491,-179.937,6.344,149.133
C04177=1144.250,37.038,-50.476,-179.940,6.344,149.134
C04178=1144.254,36.789,-50.461,-179.942,6.343,149.134
C04179=1144.259,36.539,-50.447,-179.944,6.341,149.135
C04180=1144.265,36.290,-50.431,-179.947,6.341,149.135
C04181=1144.270,36.040,-50.417,-179.950,6.339,149.136
C04182=1144.274,35.791,-50.402,-179.952,6.338,149.136
C04183=1144.280,35.541,-50.387,-179.955,6.338,149.137
C04184=1144.285,35.292,-50.372,-179.957,6.336,149.137
C04185=1144.290,35.043,-50.357,-179.960,6.336,149.138
C04186=1144.295,34.793,-50.342,-179.963,6.334,149.139
C04187=1144.300,34.543,-50.328,-179.965,6.333,149.139
C04188=1144.305,34.294,-50.313,-179.968,6.332,149.140
C04189=1144.310,34.044,-50.298,-179.970,6.331,149.140
C04190=1144.315,33.795,-50.283,-179.973,6.331,149.141
C04191=1144.321,33.545,-50.268,-179.976,6.329,149.141
C04192=1144.325,33.296,-50.253,-179.978,6.328,149.142
C04193=1144.330,33.046,-50.239,-179.981,6.327,149.142
C04194=1144.335,32.797,-50.224,-179.983,6.326,149.143
C04195=1144.341,32.547,-50.209,-179.986,6.326,149.144
C04196=1144.346,32.297,-50.195,-179.989,6.324,149.144
C04197=1144.350,32.048,-50.180,-179.991,6.323,149.144
C04198=1144.355,31.799,-50.166,-179.994,6.323,149.145
C04199=1144.361,31.549,-50.150,-179.996,6.321,149.146
C04200=1144.366,31.299,-50.136,-179.999,6.321,149.146
C04201=1144.371,31.050,-50.122,179.998,6.319,149.147
C04202=1144.375,30.801,-50.107,179.996,6.318,149.147
C04203=1144.381,30.551,-50.092,179.993,6.318,149.148
C04204=1144.386,30.301,-50.077,179.991,6.316,149.148
C04205=1144.390,30.052,-50.063,179.988,6.316,149.149
C04206=1144.395,29.802,-50.048,179.986,6.315,149.149
C04207=1144.402,29.553,-50.034,179.983,6.313,149.150
C04208=1144.406,29.304,-50.019,179.980,6.313,149.151
C04209=1144.411,29.054,-50.004,179.978,6.311,149.151
C04210=1144.416,28.804,-49.990,179.975,6.311,149.152
C04211=1144.421,28.555,-49.976,179.973,6.310,149.152
C04212=1144.426,28.305,-49.961,179.970,6.308,149.153
C04213=1144.432,28.055,-49.946,179.967,6.308,149.153
C04214=1144.437,27.787,-49.930,179.965,6.306,149.154
C04215=1144.442,27.517,-49.915,179.962,6.306,149.154
C04216=1144.448,27.249,-49.900,179.959,6.304,149.155
C04217=1144.454,26.980,-49.884,179.957,6.304,149.156
C04218=1144.459,26.730,-49.869,179.954,6.302,149.156
C04219=1144.464,26.481,-49.855,179.951,6.302,149.157
C04220=1144.469,26.231,-49.841,179.949,6.301,149.157
C04221=1144.474,25.981,-49.827,179.946,6.300,149.158
C04222=1144.478,25.732,-49.812,179.944,6.299,149.158
C04223=1144.484,25.483,-49.798,179.941,6.298,149.159
C04224=1144.489,25.233,-49.783,179.938,6.297,149.159
C04225=1144.494,24.984,-49.769,179.936,6.296,149.160
C04226=1144.499,24.734,-49.754,179.933,6.295,149.161
C04227=1144.504,24.484,-49.740,179.931,6.294,149.161
C04228=1144.509,24.234,-49.726,179.928,6.293,149.162
C04229=1144.514,23.986,-49.711,179.926,6.292,149.162
C04230=1144.519,23.736,-49.697,179.923,6.291,149.163
C04231=1144.524,23.486,-49.683,179.920,6.290,149.163
C04232=1144.529,23.237,-49.668,179.918,6.290,149.164
C04233=1144.534,22.987,-49.654,179.915,6.288,149.164
C04234=1144.540,22.738,-49.640,179.913,6.288,149.165
C04235=1144.545,22.488,-49.626,179.911,6.287,149.165
C04236=1144.550,22.239,-49.611,179.907,6.285,149.166
C04237=1144.555,21.989,-49.597,179.905,6.285,149.166
C04238=1144.560,21.739,-49.583,179.903,6.284,149.167
C04239=1144.565,21.490,-49.569,179.900,6.283,149.168
C04240=1144.570,21.240,-49.555,179.898,6.282,149.168
C04241=1144.575,20.991,-49.540,179.895,6.281,149.169
C04242=1144.580,20.741,-49.526,179.892,6.280,149.169
C04243=1144.586,20.492,-49.512,179.890,6.279,149.170
C04244=1144.591,20.242,-49.498,179.887,6.278,149.170
C04245=1144.596,19.993,-49.484,179.885,6.278,149.171
C04246=1144.601,19.743,-49.469,179.882,6.276,149.171
C04247=1144.606,19.494,-49.456,179.880,6.275,149.172
C04248=1144.611,19.244,-49.441,179.877,6.275,149.173
C04249=1144.616,18.994,-49.427,179.874,6.273,149.173
C04250=1144.620,18.745,-49.413,179.872,6.273,149.174
C04251=1144.626,18.495,-49.400,179.870,6.272,149.174
C04252=1144.631,18.246,-49.386,179.867,6.271,149.175
C04253=1144.636,17.996,-49.372,179.864,6.270,149.175
C04254=1144.642,17.747,-49.358,179.862,6.269,149.176
C04255=1144.646,17.497,-49.343,179.859,6.269,149.176
C04256=1144.651,17.248,-49.329,179.857,6.267,149.177
C04257=1144.656,16.998,-49.315,179.854,6.266,149.177
C04258=1144.662,16.748,-49.302,179.852,6.266,149.178
C04259=1144.667,16.498,-49.287,179.849,6.264,149.178
C04260=1144.671,16.249,-49.274,179.846,6.264,149.179
C04261=1144.677,16.000,-49.260,179.844,6.263,149.180
C04262=1144.682,15.750,-49.245,179.842,6.263,149.180
C04263=1144.687,15.501,-49.231,179.839,6.261,149.181
C04264=1144.693,15.251,-49.218,179.837,6.260,149.181
C04265=1144.698,15.001,-49.204,179.834,6.260,149.182
C04266=1144.702,14.752,-49.190,179.832,6.259,149.182
C04267=1144.707,14.503,-49.176,179.829,6.258,149.183
C04268=1144.713,14.253,-49.163,179.826,6.257,149.184
C04269=1144.718,14.003,-49.148,179.824,6.256,149.184
C04270=1144.723,13.754,-49.134,179.821,6.255,149.185
C04271=1144.727,13.504,-49.121,179.819,6.254,149.185
C04272=1144.733,13.255,-49.107,179.816,6.254,149.186
C04273=1144.738,13.005,-49.093,179.814,6.253,149.186
C04274=1144.743,12.755,-49.079,179.811,6.251,149.187
C04275=1144.749,12.506,-49.066,179.809,6.251,149.187
C04276=1144.753,12.256,-49.052,179.806,6.250,149.188
C04277=1144.758,12.007,-49.038,179.804,6.249,149.189
C04278=1144.764,11.757,-49.025,179.801,6.248,149.189
C04279=1144.769,11.507,-49.010,179.798,6.247,149.190
C04280=1144.774,11.259,-48.997,179.796,6.247,149.190
C04281=1144.779,11.008,-48.983,179.793,6.246,149.191
C04282=1144.784,10.759,-48.969,179.791,6.244,149.191
C04283=1144.790,10.510,-48.955,179.788,6.244,149.192
C04284=1144.794,10.260,-48.942,179.786,6.243,149.192
C04285=1144.800,10.011,-48.928,179.784,6.242,149.193
C04286=1144.805,9.760,-48.915,179.780,6.241,149.194
C04287=1144.810,9.512,-48.901,179.778,6.240,149.194
C04288=1144.815,9.261,-48.888,179.776,6.240,149.195
C04289=1144.820,9.011,-48.874,179.773,6.239,149.195
C04290=1144.825,8.763,-48.860,179.771,6.237,149.196
C04291=1144.830,8.512,-48.847,179.768,6.237,149.196
C04292=1144.836,8.263,-48.833,179.766,6.236,149.197
C04293=1144.840,8.013,-48.820,179.763,6.236,149.198
C04294=1144.846,7.764,-48.806,179.761,6.235,149.198
C04295=1144.851,7.514,-48.792,179.758,6.233,149.198
C04296=1144.856,7.265,-48.779,179.756,6.233,149.199
C04297=1144.861,7.015,-48.766,179.753,6.232,149.200
C04298=1144.867,6.766,-48.752,179.751,6.232,149.200
C04299=1144.871,6.516,-48.739,179.748,6.230,149.201
C04300=1144.876,6.266,-48.724,179.745,6.230,149.201
C04301=1144.881,6.017,-48.712,179.743,6.229,149.202
C04302=1144.886,5.767,-48.698,179.741,6.228,149.202
C04303=1144.892,5.518,-48.684,179.738,6.228,149.203
C04304=1144.897,5.268,-48.671,179.736,6.226,149.203
C04305=1144.902,5.019,-48.657,179.733,6.226,149.204
C04306=1144.907,4.769,-48.644,179.731,6.225,149.205
C04307=1144.912,4.520,-48.631,179.729,6.224,149.205
C04308=1144.918,4.269,-48.617,179.726,6.223,149.206
C04309=1144.923,4.020,-48.604,179.723,6.222,149.206
C04310=1144.928,3.771,-48.590,179.720,6.221,149.207
C04311=1144.933,3.521,-48.578,179.718,6.221,149.207
C04312=1144.938,3.272,-48.564,179.716,6.220,149.208
C04313=1144.943,3.022,-48.551,179.713,6.219,149.209
C04314=1144.949,2.772,-48.537,179.711,6.218,149.209
C04315=1144.953,2.523,-48.524,179.708,6.217,149.210
C04316=1144.959,2.273,-48.511,179.706,6.216,149.210
C04317=1144.963,2.023,-48.498,179.703,6.216,149.211
C04318=1144.969,1.755,-48.483,179.700,6.214,149.211
C04319=1144.975,1.484,-48.469,179.698,6.214,149.212
C04320=1144.980,1.215,-48.454,179.695,6.214,149.213
C04321=1144.985,0.945,-48.440,179.692,6.212,149.213
C04322=1144.991,0.696,-48.427,179.690,6.212,149.214
C04323=1144.996,0.447,-48.414,179.688,6.211,149.214
C04324=1145.001,0.197,-48.400,179.685,6.210,149.215
C04325=1145.007,-0.053,-48.387,179.683,6.209,149.215
C04326=1145.011,-0.303,-48.374,179.680,6.208,149.216
C04327=1145.017,-0.552,-48.360,179.677,6.207,149.217
C04328=1145.022,-0.801,-48.348,179.675,6.207,149.217
C04329=1145.027,-1.051,-48.334,179.672,6.206,149.218
C04330=1145.032,-1.301,-48.322,179.670,6.205,149.218
C04331=1145.037,-1.551,-48.308,179.668,6.205,149.219
C04332=1145.042,-1.800,-48.295,179.665,6.203,149.219
C04333=1145.047,-2.049,-48.282,179.663,6.203,149.220
C04334=1145.053,-2.299,-48.269,179.660,6.202,149.221
C04335=1145.058,-2.549,-48.256,179.658,6.201,149.221
C04336=1145.064,-2.798,-48.243,179.655,6.201,149.222
C04337=1145.068,-3.048,-48.230,179.653,6.200,149.222
C04338=1145.073,-3.297,-48.217,179.650,6.198,149.223
C04339=1145.078,-3.547,-48.203,179.648,6.198,149.223
C04340=1145.083,-3.797,-48.190,179.645,6.197,149.224
C04341=1145.089,-4.046,-48.177,179.643,6.197,149.224
C04342=1145.094,-4.296,-48.164,179.641,6.196,149.225
C04343=1145.099,-4.546,-48.152,179.638,6.196,149.226
C04344=1145.105,-4.795,-48.138,179.636,6.195,149.226
C04345=1145.109,-5.045,-48.126,179.633,6.193,149.227
C04346=1145.114,-5.295,-48.113,179.630,6.193,149.227
C04347=1145.120,-5.544,-48.100,179.628,6.192,149.228
C04348=1145.124,-5.794,-48.086,179.625,6.192,149.228
C04349=1145.130,-6.043,-48.073,179.623,6.191,149.229
C04350=1145.135,-6.293,-48.060,179.621,6.190,149.230
C04351=1145.140,-6.543,-48.047,179.618,6.189,149.230
C04352=1145.145,-6.792,-48.035,179.616,6.188,149.231
C04353=1145.151,-7.041,-48.021,179.613,6.187,149.231
C04354=1145.156,-7.291,-48.009,179.611,6.187,149.232
C04355=1145.161,-7.541,-47.996,179.608,6.186,149.232
C04356=1145.166,-7.790,-47.983,179.606,6.185,149.233
C04357=1145.172,-8.040,-47.970,179.603,6.185,149.234
C04358=1145.176,-8.290,-47.957,179.601,6.184,149.234
C04359=1145.181,-8.539,-47.945,179.599,6.183,149.234
C04360=1145.187,-8.789,-47.933,179.596,6.182,149.235
C04361=1145.192,-9.039,-47.919,179.594,6.181,149.236
C04362=1145.197,-9.289,-47.906,179.591,6.181,149.236
C04363=1145.202,-9.538,-47.894,179.589,6.180,149.237
C04364=1145.207,-9.787,-47.881,179.586,6.179,149.237
C04365=1145.212,-10.037,-47.869,179.584,6.179,149.238
C04366=1145.218,-10.287,-47.855,179.582,6.178,149.238
C04367=1145.223,-10.536,-47.843,179.579,6.178,149.239
C04368=1145.228,-10.786,-47.830,179.577,6.177,149.240
C04369=1145.233,-11.035,-47.817,179.574,6.176,149.240
C04370=1145.237,-11.285,-47.804,179.571,6.175,149.241
C04371=1145.244,-11.535,-47.792,179.569,6.174,149.241
C04372=1145.249,-11.785,-47.779,179.567,6.174,149.242
C04373=1145.254,-12.034,-47.767,179.564,6.173,149.242
C04374=1145.258,-12.284,-47.754,179.562,6.172,149.243
C04375=1145.264,-12.533,-47.741,179.560,6.172,149.244
C04376=1145.269,-12.782,-47.729,179.557,6.171,149.244
C04377=1145.275,-13.033,-47.716,179.555,6.170,149.245
C04378=1145.280,-13.282,-47.703,179.553,6.170,149.245
C04379=1145.284,-13.532,-47.690,179.549,6.168,149.246
C04380=1145.290,-13.781,-47.678,179.547,6.168,149.246
C04381=1145.295,-14.031,-47.665,179.544,6.167,149.247
C04382=1145.300,-14.281,-47.653,179.542,6.166,149.247
C04383=1145.305,-14.530,-47.641,179.540,6.166,149.248
C04384=1145.310,-14.780,-47.628,179.537,6.165,149.249
C04385=1145.316,-15.030,-47.615,179.535,6.164,149.249
C04386=1145.321,-15.280,-47.603,179.533,6.164,149.250
C04387=1145.326,-15.529,-47.590,179.530,6.163,149.250
C04388=1145.331,-15.778,-47.578,179.528,6.163,149.251
C04389=1145.337,-16.028,-47.566,179.526,6.162,149.251
C04390=1145.341,-16.278,-47.553,179.523,6.161,149.252
C04391=1145.346,-16.527,-47.540,179.520,6.160,149.253
C04392=1145.352,-16.777,-47.527,179.518,6.159,149.253
C04393=1145.357,-17.027,-47.516,179.515,6.159,149.254
C04394=1145.362,-17.276,-47.503,179.513,6.158,149.254
C04395=1145.367,-17.525,-47.490,179.510,6.157,149.255
C04396=1145.373,-17.775,-47.478,179.508,6.157,149.255
C04397=1145.377,-18.025,-47.466,179.506,6.156,149.256
C04398=1145.383,-18.275,-47.454,179.503,6.155,149.257
C04399=1145.388,-18.525,-47.441,179.501,6.155,149.257
C04400=1145.393,-18.774,-47.428,179.499,6.154,149.258
C04401=1145.398,-19.024,-47.417,179.496,6.153,149.258
C04402=1145.403,-19.273,-47.404,179.494,6.153,149.259
C04403=1145.409,-19.522,-47.391,179.492,6.152,149.259
C04404=1145.414,-19.772,-47.379,179.489,6.151,149.260
C04405=1145.419,-20.022,-47.367,179.487,6.151,149.261
C04406=1145.424,-20.272,-47.355,179.485,6.150,149.261
C04407=1145.429,-20.522,-47.342,179.482,6.150,149.262
C04408=1145.434,-20.772,-47.330,179.479,6.148,149.262
C04409=1145.440,-21.021,-47.318,179.477,6.147,149.263
C04410=1145.445,-21.271,-47.306,179.474,6.147,149.263
C04411=1145.450,-21.520,-47.293,179.472,6.146,149.264
C04412=1145.456,-21.770,-47.281,179.469,6.146,149.264
C04413=1145.461,-22.019,-47.269,179.467,6.145,149.265
C04414=1145.466,-22.269,-47.257,179.465,6.144,149.266
C04415=1145.471,-22.519,-47.244,179.462,6.144,149.266
C04416=1145.477,-22.769,-47.232,179.460,6.143,149.267
C04417=1145.482,-23.018,-47.220,179.458,6.142,149.267
C04418=1145.487,-23.268,-47.208,179.455,6.142,149.268
C04419=1145.492,-23.517,-47.195,179.453,6.141,149.268
C04420=1145.498,-23.767,-47.183,179.450,6.140,149.269
C04421=1145.503,-24.016,-47.171,179.448,6.140,149.269
C04422=1145.508,-24.287,-47.158,179.446,6.139,149.270
C04423=1145.514,-24.557,-47.145,179.443,6.139,149.271
C04424=1145.519,-24.827,-47.132,179.440,6.137,149.271
C04425=1145.524,-25.096,-47.118,179.438,6.137,149.272
C04426=1145.530,-25.346,-47.107,179.435,6.136,149.272
C04427=1145.535,-25.596,-47.095,179.433,6.136,149.273
C04428=1145.540,-25.846,-47.082,179.430,6.135,149.274
C04429=1145.546,-26.096,-47.070,179.428,6.134,149.274
C04430=1145.551,-26.345,-47.058,179.426,6.134,149.275
C04431=1145.556,-26.595,-47.046,179.423,6.133,149.275
C04432=1145.561,-26.845,-47.034,179.421,6.132,149.276
C04433=1145.566,-27.094,-47.022,179.419,6.132,149.276
C04434=1145.572,-27.344,-47.010,179.416,6.131,149.277
C04435=1145.577,-27.594,-46.998,179.414,6.130,149.278
C04436=1145.582,-27.843,-46.985,179.412,6.130,149.278
C04437=1145.587,-28.093,-46.974,179.409,6.129,149.279
C04438=1145.592,-28.343,-46.962,179.407,6.128,149.279
C04439=1145.597,-28.592,-46.950,179.404,6.128,149.280
C04440=1145.603,-28.842,-46.938,179.402,6.127,149.280
C04441=1145.608,-29.091,-46.926,179.400,6.126,149.281
C04442=1145.613,-29.341,-46.914,179.397,6.126,149.282
C04443=1145.618,-29.591,-46.902,179.395,6.125,149.282
C04444=1145.624,-29.841,-46.890,179.392,6.125,149.283
C04445=1145.630,-30.090,-46.879,179.390,6.124,149.283
C04446=1145.634,-30.339,-46.867,179.387,6.124,149.284
C04447=1145.639,-30.589,-46.855,179.385,6.123,149.284
C04448=1145.645,-30.839,-46.843,179.383,6.122,149.285
C04449=1145.650,-31.088,-46.831,179.380,6.122,149.286
C04450=1145.655,-31.338,-46.820,179.378,6.121,149.286
C04451=1145.660,-31.588,-46.807,179.375,6.120,149.287
C04452=1145.666,-31.838,-46.795,179.373,6.120,149.287
C04453=1145.670,-32.087,-46.784,179.371,6.119,149.288
C04454=1145.676,-32.337,-46.772,179.368,6.118,149.288
C04455=1145.681,-32.587,-46.760,179.366,6.118,149.289
C04456=1145.685,-32.836,-46.748,179.364,6.117,149.290
C04457=1145.691,-33.085,-46.737,179.361,6.116,149.290
C04458=1145.697,-33.335,-46.725,179.359,6.116,149.291
C04459=1145.702,-33.585,-46.713,179.357,6.115,149.291
C04460=1145.707,-33.835,-46.701,179.354,6.114,149.292
C04461=1145.712,-34.085,-46.690,179.352,6.114,149.292
C04462=1145.718,-34.335,-46.678,179.350,6.113,149.293
C04463=1145.723,-34.584,-46.666,179.348,6.113,149.293
C04464=1145.728,-34.834,-46.654,179.345,6.113,149.294
C04465=1145.733,-35.083,-46.643,179.343,6.112,149.294
C04466=1145.738,-35.332,-46.631,179.340,6.112,149.295
C04467=1145.744,-35.582,-46.619,179.338,6.111,149.296
C04468=1145.749,-35.832,-46.608,179.336,6.110,149.296
C04469=1145.754,-36.082,-46.596,179.333,6.110,149.297
C04470=1145.759,-36.332,-46.584,179.331,6.109,149.297
C04471=1145.764,-36.582,-46.573,179.329,6.108,149.298
C04472=1145.770,-36.831,-46.561,179.326,6.108,149.298
C04473=1145.775,-37.080,-46.550,179.324,6.107,149.299
C04474=1145.780,-37.330,-46.538,179.322,6.106,149.300
C04475=1145.786,-37.580,-46.526,179.319,6.106,149.300
C04476=1145.790,-37.830,-46.515,179.317,6.105,149.301
C04477=1145.796,-38.080,-46.503,179.314,6.105,149.301
C04478=1145.801,-38.329,-46.492,179.312,6.104,149.302
C04479=1145.807,-38.579,-46.480,179.310,6.103,149.302
C04480=1145.812,-38.829,-46.468,179.307,6.103,149.303
C04481=1145.817,-39.078,-46.457,179.305,6.102,149.304
C04482=1145.822,-39.328,-46.445,179.303,6.101,149.304
C04483=1145.827,-39.577,-46.434,179.301,6.101,149.305
C04484=1145.833,-39.827,-46.422,179.298,6.101,149.305
C04485=1145.837,-40.077,-46.411,179.296,6.100,149.306
C04486=1145.843,-40.327,-46.399,179.293,6.100,149.306
C04487=1145.848,-40.576,-46.388,179.291,6.099,149.307
C04488=1145.854,-40.825,-46.376,179.289,6.098,149.307
C04489=1145.858,-41.075,-46.365,179.286,6.098,149.308
C04490=1145.864,-41.326,-46.354,179.284,6.097,149.309
C04491=1145.869,-41.575,-46.343,179.282,6.096,149.309
C04492=1145.875,-41.825,-46.331,179.279,6.096,149.310
C04493=1145.879,-42.074,-46.320,179.277,6.095,149.310
C04494=1145.885,-42.324,-46.308,179.275,6.095,149.311
C04495=1145.890,-42.574,-46.297,179.272,6.094,149.311
C04496=1145.896,-42.823,-46.285,179.270,6.093,149.312
C04497=1145.900,-43.073,-46.274,179.268,6.093,149.313
C04498=1145.906,-43.323,-46.263,179.266,6.093,149.313
C04499=1145.911,-43.573,-46.251,179.263,6.092,149.314
C04500=1145.917,-43.822,-46.240,179.261,6.091,149.314
C04501=1145.921,-44.072,-46.229,179.259,6.091,149.315
C04502=1145.926,-44.321,-46.217,179.256,6.090,149.315
C04503=1145.933,-44.571,-46.206,179.254,6.089,149.316
C04504=1145.937,-44.821,-46.195,179.251,6.089,149.317
C04505=1145.943,-45.071,-46.183,179.249,6.088,149.317
C04506=1145.947,-45.320,-46.172,179.247,6.088,149.318
C04507=1145.953,-45.570,-46.160,179.244,6.087,149.318
C04508=1145.958,-45.820,-46.150,179.243,6.087,149.319
C04509=1145.963,-46.069,-46.139,179.241,6.086,149.319
C04510=1145.969,-46.319,-46.127,179.238,6.086,149.320
C04511=1145.974,-46.568,-46.116,179.236,6.085,149.320
C04512=1145.979,-46.819,-46.105,179.233,6.085,149.321
C04513=1145.985,-47.068,-46.094,179.231,6.084,149.322
C04514=1145.989,-47.317,-46.082,179.229,6.083,149.322
C04515=1145.995,-47.568,-46.071,179.226,6.083,149.323
C04516=1146.001,-47.817,-46.060,179.224,6.082,149.323
C04517=1146.005,-48.066,-46.049,179.222,6.082,149.324
C04518=1146.011,-48.316,-46.037,179.220,6.082,149.324
C04519=1146.016,-48.566,-46.027,179.217,6.081,149.325
C04520=1146.021,-48.816,-46.016,179.215,6.080,149.326
C04521=1146.026,-49.066,-46.004,179.213,6.080,149.326
C04522=1146.032,-49.315,-45.994,179.210,6.079,149.327
C04523=1146.037,-49.565,-45.982,179.208,6.079,149.327
C04524=1146.042,-49.815,-45.970,179.205,6.078,149.328
C04525=1146.048,-50.064,-45.960,179.203,6.077,149.328
C04526=1146.053,-50.335,-45.948,179.201,6.077,149.329
C04527=1146.059,-50.606,-45.936,179.198,6.076,149.330
C04528=1146.065,-50.876,-45.924,179.196,6.075,149.330
C04529=1146.070,-51.147,-45.912,179.193,6.075,149.331
C04530=1146.075,-51.397,-45.900,179.191,6.074,149.331
C04531=1146.081,-51.647,-45.890,179.189,6.074,149.332
C04532=1146.086,-51.896,-45.879,179.187,6.074,149.332
C04533=1146.091,-52.146,-45.869,179.184,6.073,149.333
C04534=1146.097,-52.396,-45.857,179.182,6.073,149.334
C04535=1146.102,-52.646,-45.846,179.180,6.072,149.334
C04536=1146.107,-52.895,-45.835,179.177,6.071,149.335
C04537=1146.112,-53.144,-45.824,179.175,6.071,149.335
C04538=1146.118,-53.394,-45.813,179.173,6.071,149.336
C04539=1146.123,-53.644,-45.802,179.171,6.070,149.336
C04540=1146.128,-53.894,-45.791,179.168,6.070,149.337
C04541=1146.133,-54.143,-45.780,179.166,6.069,149.337
C04542=1146.139,-54.394,-45.769,179.163,6.068,149.338
C04543=1146.144,-54.643,-45.758,179.161,6.068,149.339
C04544=1146.149,-54.893,-45.748,179.159,6.067,149.339
C04545=1146.154,-55.142,-45.737,179.157,6.067,149.340
C04546=1146.159,-55.392,-45.726,179.155,6.066,149.340
C04547=1146.164,-55.642,-45.715,179.153,6.066,149.341
C04548=1146.170,-55.891,-45.704,179.150,6.065,149.342
C04549=1146.175,-56.141,-45.693,179.148,6.064,149.342
C04550=1146.181,-56.391,-45.683,179.146,6.064,149.342
C04551=1146.186,-56.641,-45.672,179.143,6.064,149.343
C04552=1146.191,-56.890,-45.661,179.141,6.063,149.344
C04553=1146.196,-57.140,-45.650,179.139,6.063,149.344
C04554=1146.202,-57.389,-45.639,179.136,6.062,149.345
C04555=1146.207,-57.640,-45.628,179.134,6.061,149.345
C04556=1146.212,-57.890,-45.618,179.132,6.061,149.346
C04557=1146.217,-58.139,-45.607,179.130,6.061,149.346
C04558=1146.222,-58.389,-45.596,179.128,6.060,149.347
C04559=1146.228,-58.638,-45.585,179.125,6.060,149.348
C04560=1146.233,-58.888,-45.575,179.123,6.059,149.348
C04561=1146.238,-59.138,-45.565,179.121,6.058,149.349
C04562=1146.244,-59.388,-45.553,179.118,6.058,149.349
C04563=1146.249,-59.637,-45.542,179.117,6.058,149.350
C04564=1146.254,-59.887,-45.532,179.114,6.057,149.350
C04565=1146.259,-60.136,-45.521,179.112,6.057,149.351
C04566=1146.264,-60.387,-45.510,179.109,6.056,149.351
C04567=1146.270,-60.636,-45.500,179.107,6.055,149.352
C04568=1146.275,-60.886,-45.489,179.105,6.055,149.353
C04569=1146.280,-61.135,-45.479,179.103,6.055,149.353
C04570=1146.285,-61.386,-45.468,179.101,6.054,149.354
C04571=1146.291,-61.634,-45.457,179.098,6.054,149.354
C04572=1146.296,-61.885,-45.447,179.096,6.053,149.355
C04573=1146.301,-62.134,-45.436,179.094,6.052,149.355
C04574=1146.306,-62.384,-45.426,179.092,6.053,149.356
C04575=1146.312,-62.633,-45.415,179.090,6.052,149.356
C04576=1146.318,-62.883,-45.404,179.087,6.051,149.357
C04577=1146.323,-63.133,-45.394,179.085,6.051,149.358
C04578=1146.328,-63.383,-45.383,179.082,6.050,149.358
C04579=1146.333,-63.633,-45.372,179.081,6.050,149.359
C04580=1146.339,-63.882,-45.362,179.078,6.049,149.359
C04581=1146.344,-64.132,-45.351,179.076,6.049,149.360
C04582=1146.349,-64.382,-45.341,179.074,6.048,149.360
C04583=1146.354,-64.632,-45.330,179.071,6.048,149.361
C04584=1146.360,-64.881,-45.320,179.070,6.048,149.361
C04585=1146.365,-65.131,-45.309,179.067,6.047,149.362
C04586=1146.370,-65.381,-45.299,179.065,6.046,149.363
C04587=1146.376,-65.630,-45.289,179.062,6.046,149.363
C04588=1146.381,-65.881,-45.278,179.060,6.045,149.364
C04589=1146.386,-66.130,-45.267,179.058,6.045,149.364
C04590=1146.391,-66.379,-45.257,179.056,6.044,149.365
C04591=1146.396,-66.629,-45.247,179.054,6.044,149.365
C04592=1146.402,-66.879,-45.237,179.051,6.043,149.366
C04593=1146.407,-67.129,-45.226,179.049,6.043,149.366
C04594=1146.412,-67.378,-45.216,179.047,6.043,149.367
C04595=1146.418,-67.628,-45.206,179.045,6.042,149.368
C04596=1146.423,-67.878,-45.195,179.043,6.041,149.368
C04597=1146.428,-68.127,-45.184,179.040,6.041,149.369
C04598=1146.433,-68.377,-45.174,179.038,6.041,149.369
C04599=1146.439,-68.627,-45.163,179.036,6.040,149.370
C04600=1146.444,-68.877,-45.153,179.034,6.039,149.370
C04601=1146.449,-69.127,-45.143,179.031,6.039,149.371
C04602=1146.455,-69.376,-45.132,179.029,6.038,149.372
C04603=1146.460,-69.626,-45.122,179.027,6.038,149.372
C04604=1146.465,-69.876,-45.112,179.025,6.038,149.373
C04605=1146.470,-70.125,-45.102,179.023,6.037,149.373
C04606=1146.476,-70.375,-45.092,179.020,6.036,149.374
C04607=1146.481,-70.625,-45.081,179.018,6.037,149.374
C04608=1146.487,-70.875,-45.071,179.016,6.036,149.375
C04609=1146.492,-71.124,-45.061,179.014,6.035,149.375
C04610=1146.497,-71.374,-45.050,179.011,6.035,149.376
C04611=1146.503,-71.624,-45.040,179.010,6.035,149.376
C04612=1146.508,-71.874,-45.030,179.007,6.034,149.377
C04613=1146.513,-72.123,-45.020,179.005,6.034,149.378
C04614=1146.518,-72.373,-45.010,179.003,6.033,149.378
C04615=1146.524,-72.623,-44.999,179.000,6.032,149.379
C04616=1146.529,-72.873,-44.989,178.999,6.032,149.379
C04617=1146.534,-73.122,-44.979,178.996,6.032,149.380
C04618=1146.540,-73.372,-44.968,178.994,6.031,149.380
C04619=1146.544,-73.622,-44.958,178.992,6.030,149.381
C04620=1146.550,-73.871,-44.948,178.990,6.031,149.382
C04621=1146.555,-74.121,-44.938,178.988,6.030,149.382
C04622=1146.560,-74.371,-44.927,178.985,6.029,149.382
C04623=1146.566,-74.621,-44.917,178.983,6.029,149.383
C04624=1146.571,-74.871,-44.908,178.981,6.029,149.384
C04625=1146.577,-75.120,-44.898,178.979,6.028,149.384
C04626=1146.582,-75.370,-44.888,178.977,6.027,149.385
C04627=1146.587,-75.620,-44.877,178.975,6.028,149.385
C04628=1146.593,-75.869,-44.867,178.972,6.027,149.386
C04629=1146.598,-76.119,-44.858,178.970,6.026,149.386
C04630=1146.604,-76.390,-44.846,178.968,6.026,149.387
C04631=1146.609,-76.662,-44.836,178.965,6.025,149.388
C04632=1146.615,-76.934,-44.824,178.963,6.025,149.388
C04633=1146.621,-77.204,-44.814,178.960,6.024,149.389
C04634=1146.627,-77.454,-44.803,178.958,6.024,149.389
C04635=1146.632,-77.704,-44.793,178.956,6.024,149.390
C04636=1146.637,-77.954,-44.784,178.954,6.023,149.390
C04637=1146.642,-78.204,-44.774,178.952,6.023,149.391
C04638=1146.648,-78.453,-44.764,178.950,6.022,149.392
C04639=1146.653,-78.703,-44.753,178.948,6.022,149.392
C04640=1146.658,-78.953,-44.743,178.945,6.021,149.393
C04641=1146.664,-79.203,-44.734,178.943,6.021,149.393
C04642=1146.669,-79.452,-44.724,178.941,6.021,149.394
C04643=1146.674,-79.702,-44.714,178.939,6.020,149.394
C04644=1146.679,-79.952,-44.703,178.937,6.020,149.395
C04645=1146.685,-80.202,-44.694,178.935,6.019,149.395
C04646=1146.691,-80.451,-44.684,178.932,6.019,149.396
C04647=1146.696,-80.701,-44.674,178.930,6.018,149.396
C04648=1146.701,-80.951,-44.664,178.928,6.018,149.397
C04649=1146.706,-81.201,-44.654,178.926,6.018,149.398
C04650=1146.711,-81.450,-44.644,178.924,6.017,149.398
C04651=1146.717,-81.700,-44.634,178.922,6.017,149.399
C04652=1146.722,-81.950,-44.625,178.920,6.016,149.399
C04653=1146.727,-82.200,-44.615,178.917,6.016,149.400
C04654=1146.733,-82.450,-44.605,178.915,6.015,149.400
C04655=1146.737,-82.699,-44.595,178.913,6.015,149.401
C04656=1146.743,-82.949,-44.585,178.911,6.015,149.401
C04657=1146.749,-83.198,-44.575,178.909,6.014,149.402
C04658=1146.754,-83.448,-44.566,178.907,6.014,149.402
C04659=1146.759,-83.699,-44.556,178.904,6.013,149.403
C04660=1146.765,-83.948,-44.546,178.902,6.013,149.404
C04661=1146.770,-84.197,-44.536,178.900,6.012,149.404
C04662=1146.776,-84.447,-44.526,178.898,6.012,149.405
C04663=1146.780,-84.697,-44.517,178.896,6.012,149.405
C04664=1146.786,-84.947,-44.507,178.894,6.011,149.406
C04665=1146.791,-85.197,-44.497,178.892,6.011,149.406
C04666=1146.796,-85.446,-44.487,178.889,6.010,149.407
C04667=1146.802,-85.697,-44.478,178.887,6.010,149.407
C04668=1146.807,-85.946,-44.468,178.886,6.010,149.408
C04669=1146.813,-86.196,-44.459,178.883,6.009,149.408
C04670=1146.818,-86.445,-44.449,178.881,6.009,149.409
C04671=1146.823,-86.695,-44.439,178.879,6.009,149.410
C04672=1146.828,-86.945,-44.429,178.877,6.008,149.410
C04673=1146.833,-87.195,-44.419,178.875,6.007,149.411
C04674=1146.839,-87.445,-44.410,178.873,6.008,149.411
C04675=1146.844,-87.694,-44.400,178.870,6.007,149.412
C04676=1146.849,-87.944,-44.391,178.868,6.006,149.412
C04677=1146.855,-88.194,-44.381,178.866,6.005,149.413
C04678=1146.860,-88.443,-44.372,178.864,6.006,149.413
C04679=1146.866,-88.693,-44.362,178.862,6.005,149.414
C04680=1146.871,-88.942,-44.352,178.860,6.004,149.414
C04681=1146.876,-89.193,-44.342,178.858,6.004,149.415
C04682=1146.881,-89.442,-44.333,178.855,6.004,149.416
C04683=1146.887,-89.692,-44.323,178.853,6.003,149.416
C04684=1146.892,-89.942,-44.314,178.851,6.003,149.417
C04685=1146.897,-90.192,-44.304,178.849,6.002,149.417
C04686=1146.903,-90.442,-44.295,178.847,6.002,149.418
C04687=1146.908,-90.691,-44.285,178.845,6.002,149.418
C04688=1146.913,-90.941,-44.276,178.843,6.001,149.419
C04689=1146.919,-91.191,-44.266,178.841,6.000,149.419
C04690=1146.924,-91.440,-44.257,178.839,6.001,149.420
C04691=1146.930,-91.690,-44.247,178.836,6.000,149.420
C04692=1146.935,-91.940,-44.238,178.834,5.999,149.421
C04693=1146.940,-92.189,-44.228,178.833,5.999,149.421
C04694=1146.946,-92.439,-44.219,178.830,5.999,149.422
C04695=1146.951,-92.689,-44.210,178.828,5.998,149.423
C04696=1146.956,-92.939,-44.199,178.826,5.998,149.423
C04697=1146.961,-93.189,-44.191,178.824,5.997,149.423
C04698=1146.967,-93.439,-44.180,178.822,5.998,149.424
C04699=1146.972,-93.689,-44.171,178.820,5.997,149.425
C04700=1146.978,-93.939,-44.162,178.817,5.996,149.425
C04701=1146.983,-94.188,-44.152,178.816,5.996,149.426
C04702=1146.988,-94.438,-44.143,178.814,5.996,149.426
C04703=1146.993,-94.687,-44.133,178.811,5.995,149.427
C04704=1146.998,-94.937,-44.124,178.809,5.995,149.427
C04705=1147.004,-95.187,-44.115,178.807,5.995,149.428
C04706=1147.009,-95.437,-44.105,178.805,5.994,149.428
C04707=1147.014,-95.687,-44.096,178.803,5.994,149.429
C04708=1147.020,-95.937,-44.087,178.801,5.993,149.430
C04709=1147.025,-96.186,-44.077,178.799,5.993,149.430
C04710=1147.030,-96.436,-44.068,178.797,5.993,149.430
C04711=1147.036,-96.686,-44.059,178.795,5.992,149.431
C04712=1147.041,-96.936,-44.050,178.793,5.992,149.432
C04713=1147.047,-97.185,-44.040,178.790,5.992,149.432
C04714=1147.052,-97.435,-44.031,178.788,5.991,149.433
C04715=1147.057,-97.685,-44.022,178.787,5.991,149.433
C04716=1147.063,-97.935,-44.012,178.784,5.990,149.434
C04717=1147.068,-98.184,-44.003,178.782,5.990,149.434
C04718=1147.073,-98.434,-43.994,178.780,5.990,149.435
C04719=1147.079,-98.684,-43.984,178.778,5.989,149.435
C04720=1147.084,-98.934,-43.975,178.776,5.988,149.436
C04721=1147.090,-99.183,-43.966,178.774,5.988,149.436
C04722=1147.096,-99.433,-43.957,178.772,5.988,149.437
C04723=1147.101,-99.683,-43.948,178.770,5.988,149.437
C04724=1147.106,-99.932,-43.938,178.768,5.987,149.438
C04725=1147.111,-100.182,-43.929,178.766,5.987,149.438
C04726=1147.117,-100.432,-43.920,178.764,5.987,149.439
C04727=1147.122,-100.682,-43.911,178.761,5.986,149.440
C04728=1147.127,-100.932,-43.902,178.759,5.985,149.440
C04729=1147.133,-101.181,-43.892,178.758,5.985,149.441
C04730=1147.138,-101.431,-43.883,178.755,5.985,149.441
C04731=1147.143,-101.681,-43.874,178.754,5.985,149.442
C04732=1147.148,-101.931,-43.865,178.751,5.984,149.442
C04733=1147.154,-102.181,-43.856,178.749,5.984,149.443
C04734=1147.160,-102.453,-43.846,178.747,5.984,149.443
C04735=1147.166,-102.725,-43.836,178.745,5.983,149.444
C04736=1147.171,-102.997,-43.826,178.742,5.983,149.444
C04737=1147.177,-103.269,-43.817,178.740,5.982,149.445
C04738=1147.182,-103.518,-43.807,178.738,5.982,149.446
C04739=1147.187,-103.768,-43.798,178.736,5.981,149.446
C04740=1147.193,-104.019,-43.789,178.734,5.981,149.447
C04741=1147.198,-104.268,-43.780,178.732,5.981,149.447
C04742=1147.204,-104.518,-43.771,178.730,5.980,149.448
C04743=1147.209,-104.768,-43.762,178.728,5.980,149.448
C04744=1147.215,-105.018,-43.753,178.726,5.980,149.449
C04745=1147.220,-105.267,-43.744,178.724,5.980,149.449
C04746=1147.226,-105.517,-43.735,178.722,5.979,149.450
C04747=1147.231,-105.767,-43.726,178.720,5.978,149.450
C04748=1147.236,-106.016,-43.716,178.718,5.978,149.451
C04749=1147.241,-106.266,-43.708,178.716,5.977,149.451
C04750=1147.247,-106.516,-43.698,178.714,5.978,149.452
C04751=1147.252,-106.766,-43.689,178.712,5.977,149.452
C04752=1147.258,-107.015,-43.681,178.709,5.976,149.453
C04753=1147.263,-107.265,-43.672,178.708,5.976,149.453
C04754=1147.268,-107.515,-43.663,178.706,5.976,149.454
C04755=1147.273,-107.765,-43.654,178.704,5.976,149.455
C04756=1147.278,-108.015,-43.645,178.701,5.975,149.455
C04757=1147.284,-108.265,-43.636,178.699,5.975,149.456
C04758=1147.289,-108.515,-43.627,178.698,5.975,149.456
C04759=1147.295,-108.764,-43.618,178.695,5.974,149.457
C04760=1147.300,-109.014,-43.609,178.694,5.974,149.457
C04761=1147.305,-109.264,-43.600,178.692,5.973,149.458
C04762=1147.311,-109.513,-43.591,178.689,5.974,149.458
C04763=1147.316,-109.763,-43.583,178.687,5.973,149.459
C04764=1147.322,-110.012,-43.574,178.685,5.972,149.459
C04765=1147.327,-110.263,-43.565,178.683,5.972,149.460
C04766=1147.333,-110.512,-43.556,178.681,5.971,149.460
C04767=1147.338,-110.763,-43.547,178.680,5.971,149.461
C04768=1147.343,-111.013,-43.539,178.677,5.971,149.461
C04769=1147.348,-111.263,-43.530,178.675,5.971,149.462
C04770=1147.354,-111.512,-43.521,178.673,5.970,149.462
C04771=1147.359,-111.762,-43.512,178.671,5.970,149.463
C04772=1147.365,-112.011,-43.503,178.669,5.970,149.463
C04773=1147.370,-112.261,-43.494,178.667,5.969,149.464
C04774=1147.375,-112.511,-43.486,178.666,5.969,149.464
C04775=1147.381,-112.760,-43.477,178.663,5.969,149.465
C04776=1147.386,-113.010,-43.468,178.661,5.969,149.465
C04777=1147.391,-113.260,-43.459,178.659,5.968,149.466
C04778=1147.396,-113.511,-43.451,178.657,5.967,149.466
C04779=1147.402,-113.760,-43.442,178.655,5.967,149.467
C04780=1147.408,-114.010,-43.433,178.653,5.966,149.467
C04781=1147.413,-114.260,-43.424,178.652,5.966,149.468
C04782=1147.418,-114.510,-43.415,178.649,5.966,149.468
C04783=1147.424,-114.759,-43.407,178.647,5.966,149.469
C04784=1147.430,-115.009,-43.398,178.645,5.965,149.470
C04785=1147.435,-115.259,-43.390,178.644,5.965,149.470
C04786=1147.440,-115.509,-43.381,178.641,5.965,149.471
C04787=1147.446,-115.758,-43.372,178.639,5.964,149.471
C04788=1147.451,-116.008,-43.363,178.638,5.964,149.472
C04789=1147.456,-116.258,-43.354,178.635,5.963,149.472
C04790=1147.462,-116.508,-43.346,178.634,5.963,149.473
C04791=1147.467,-116.757,-43.338,178.631,5.963,149.473
C04792=1147.472,-117.007,-43.329,178.629,5.963,149.474
C04793=1147.478,-117.257,-43.320,178.627,5.962,149.474
C04794=1147.483,-117.508,-43.312,178.626,5.962,149.475
C04795=1147.489,-117.757,-43.303,178.623,5.961,149.475
C04796=1147.493,-118.006,-43.295,178.622,5.961,149.476
C04797=1147.498,-118.256,-43.286,178.620,5.961,149.476
C04798=1147.505,-118.506,-43.278,178.617,5.960,149.477
C04799=1147.510,-118.756,-43.269,178.616,5.960,149.477
C04800=1147.515,-119.006,-43.260,178.613,5.960,149.478
C04801=1147.520,-119.255,-43.251,178.612,5.960,149.478
C04802=1147.526,-119.505,-43.244,178.609,5.959,149.479
C04803=1147.531,-119.755,-43.235,178.608,5.959,149.479
C04804=1147.536,-120.005,-43.226,178.606,5.958,149.480
C04805=1147.543,-120.255,-43.218,178.604,5.958,149.480
C04806=1147.548,-120.504,-43.209,178.602,5.958,149.481
C04807=1147.553,-120.754,-43.200,178.600,5.958,149.481
C04808=1147.559,-121.003,-43.192,178.598,5.957,149.482
C04809=1147.563,-121.254,-43.184,178.596,5.957,149.482
C04810=1147.569,-121.503,-43.175,178.594,5.956,149.483
C04811=1147.574,-121.753,-43.167,178.592,5.957,149.483
C04812=1147.580,-122.003,-43.158,178.590,5.956,149.484
C04813=1147.585,-122.253,-43.150,178.588,5.956,149.484
C04814=1147.590,-122.503,-43.141,178.586,5.955,149.485
C04815=1147.596,-122.753,-43.133,178.584,5.954,149.485
C04816=1147.601,-123.002,-43.124,178.582,5.954,149.486
C04817=1147.607,-123.252,-43.117,178.580,5.954,149.486
C04818=1147.612,-123.502,-43.108,178.579,5.954,149.487
C04819=1147.617,-123.752,-43.099,178.576,5.953,149.487
C04820=1147.623,-124.001,-43.091,178.575,5.953,149.488
C04821=1147.628,-124.251,-43.082,178.573,5.952,149.488
C04822=1147.634,-124.502,-43.074,178.571,5.953,149.489
C04823=1147.639,-124.751,-43.066,178.568,5.952,149.490
C04824=1147.644,-125.000,-43.057,178.567,5.952,149.490
C04825=1147.649,-125.251,-43.049,178.565,5.951,149.491
C04826=1147.655,-125.500,-43.041,178.563,5.951,149.491
C04827=1147.661,-125.750,-43.032,178.561,5.950,149.491
C04828=1147.666,-126.000,-43.023,178.559,5.951,149.492
C04829=1147.671,-126.250,-43.016,178.557,5.950,149.492
C04830=1147.676,-126.500,-43.007,178.555,5.950,149.493
C04831=1147.682,-126.749,-42.999,178.553,5.949,149.493
C04832=1147.688,-126.999,-42.991,178.552,5.949,149.494
C04833=1147.693,-127.249,-42.982,178.549,5.948,149.494
C04834=1147.698,-127.499,-42.974,178.548,5.948,149.495
C04835=1147.703,-127.748,-42.966,178.546,5.948,149.495
C04836=1147.709,-127.998,-42.958,178.544,5.948,149.496
C04837=1147.714,-128.248,-42.949,178.542,5.947,149.496
C04838=1147.294,-128.259,-42.992,178.539,5.951,149.498
C04839=1147.288,-128.010,-43.000,178.540,5.951,149.498
C04840=1147.283,-127.760,-43.009,178.542,5.952,149.497
C04841=1147.277,-127.510,-43.017,178.544,5.952,149.497
C04842=1147.272,-127.260,-43.026,178.546,5.952,149.496
C04843=1147.267,-127.010,-43.033,178.548,5.952,149.496
C04844=1147.261,-126.761,-43.042,178.550,5.953,149.495
C04845=1147.256,-126.510,-43.050,178.551,5.953,149.495
C04846=1147.250,-126.261,-43.059,178.554,5.954,149.494
C04847=1147.244,-126.011,-43.067,178.555,5.954,149.494
C04848=1147.240,-125.761,-43.075,178.557,5.955,149.493
C04849=1147.234,-125.511,-43.083,178.559,5.955,149.493
C04850=1147.229,-125.262,-43.092,178.561,5.955,149.492
C04851=1147.224,-125.012,-43.101,178.563,5.955,149.492
C04852=1147.218,-124.762,-43.109,178.566,5.956,149.491
C04853=1147.213,-124.512,-43.117,178.567,5.956,149.491
C04854=1147.207,-124.263,-43.125,178.569,5.956,149.490
C04855=1147.202,-124.013,-43.134,178.571,5.956,149.490
C04856=1147.197,-123.763,-43.142,178.573,5.957,149.489
C04857=1147.191,-123.513,-43.150,178.575,5.957,149.489
C04858=1147.185,-123.263,-43.159,178.577,5.958,149.488
C04859=1147.180,-123.013,-43.167,178.579,5.958,149.488
C04860=1147.175,-122.764,-43.175,178.581,5.958,149.487
C04861=1147.170,-122.514,-43.184,178.582,5.958,149.487
C04862=1147.164,-122.264,-43.192,178.585,5.959,149.486
C04863=1147.159,-122.015,-43.201,178.586,5.959,149.486
C04864=1147.153,-121.765,-43.210,178.589,5.959,149.485
C04865=1147.148,-121.514,-43.218,178.591,5.960,149.485
C04866=1147.142,-121.265,-43.227,178.593,5.960,149.484
C04867=1147.137,-121.015,-43.235,178.595,5.961,149.484
C04868=1147.132,-120.765,-43.243,178.596,5.961,149.483
C04869=1147.126,-120.516,-43.252,178.599,5.962,149.483
C04870=1147.121,-120.266,-43.260,178.600,5.962,149.482
C04871=1147.116,-120.016,-43.269,178.602,5.962,149.482
C04872=1147.111,-119.766,-43.278,178.604,5.962,149.481
C04873=1147.105,-119.517,-43.286,178.606,5.963,149.481
C04874=1147.099,-119.266,-43.294,178.608,5.963,149.480
C04875=1147.094,-119.016,-43.303,178.610,5.963,149.479
C04876=1147.088,-118.767,-43.312,178.612,5.963,149.479
C04877=1147.083,-118.517,-43.321,178.614,5.964,149.478
C04878=1147.078,-118.267,-43.329,178.616,5.964,149.478
C04879=1147.072,-118.018,-43.337,178.618,5.965,149.478
C04880=1147.067,-117.768,-43.346,178.620,5.965,149.477
C04881=1147.062,-117.518,-43.355,178.622,5.965,149.477
C04882=1147.057,-117.268,-43.363,178.624,5.966,149.476
C04883=1147.051,-117.019,-43.371,178.626,5.966,149.476
C04884=1147.046,-116.769,-43.380,178.628,5.966,149.475
C04885=1147.041,-116.519,-43.389,178.630,5.966,149.474
C04886=1147.035,-116.269,-43.397,178.632,5.967,149.474
C04887=1147.030,-116.019,-43.406,178.634,5.967,149.473
C04888=1147.025,-115.770,-43.415,178.636,5.968,149.473
C04889=1147.019,-115.520,-43.424,178.637,5.968,149.472
C04890=1147.014,-115.271,-43.432,178.640,5.969,149.472
C04891=1147.008,-115.021,-43.441,178.642,5.969,149.471
C04892=1147.003,-114.770,-43.449,178.643,5.969,149.471
C04893=1146.998,-114.520,-43.458,178.646,5.970,149.470
C04894=1146.993,-114.270,-43.467,178.648,5.970,149.470
C04895=1146.986,-114.021,-43.476,178.650,5.970,149.469
C04896=1146.981,-113.771,-43.485,178.652,5.970,149.469
C04897=1146.976,-113.521,-43.494,178.654,5.971,149.468
C04898=1146.970,-113.271,-43.502,178.656,5.972,149.468
C04899=1146.965,-113.022,-43.511,178.658,5.972,149.467
C04900=1146.959,-112.772,-43.519,178.660,5.973,149.467
C04901=1146.954,-112.522,-43.528,178.662,5.972,149.466
C04902=1146.949,-112.272,-43.537,178.664,5.973,149.466
C04903=1146.943,-112.023,-43.546,178.666,5.973,149.465
C04904=1146.938,-111.773,-43.555,178.668,5.974,149.465
C04905=1146.933,-111.523,-43.564,178.669,5.974,149.464
C04906=1146.928,-111.273,-43.572,178.672,5.974,149.464
C04907=1146.922,-111.023,-43.581,178.674,5.975,149.463
C04908=1146.917,-110.774,-43.589,178.676,5.975,149.462
C04909=1146.911,-110.524,-43.598,178.678,5.975,149.462
C04910=1146.906,-110.274,-43.607,178.680,5.975,149.462
C04911=1146.900,-110.024,-43.616,178.682,5.976,149.461
C04912=1146.895,-109.774,-43.625,178.683,5.976,149.461
C04913=1146.890,-109.524,-43.634,178.686,5.977,149.460
C04914=1146.884,-109.275,-43.643,178.688,5.978,149.460
C04915=1146.879,-109.025,-43.652,178.690,5.977,149.459
C04916=1146.874,-108.775,-43.661,178.692,5.978,149.458
C04917=1146.869,-108.526,-43.670,178.694,5.978,149.458
C04918=1146.864,-108.276,-43.678,178.696,5.979,149.457
C04919=1146.858,-108.026,-43.688,178.698,5.979,149.457
C04920=1146.852,-107.776,-43.696,178.700,5.979,149.456
C04921=1146.847,-107.527,-43.705,178.702,5.980,149.456
C04922=1146.842,-107.277,-43.714,178.704,5.980,149.455
C04923=1146.836,-107.027,-43.723,178.706,5.980,149.455
C04924=1146.831,-106.777,-43.732,178.708,5.980,149.454
C04925=1146.826,-106.527,-43.741,178.710,5.981,149.454
C04926=1146.820,-106.277,-43.750,178.712,5.982,149.453
C04927=1146.814,-106.028,-43.759,178.714,5.981,149.453
C04928=1146.809,-105.778,-43.768,178.716,5.982,149.452
C04929=1146.804,-105.528,-43.777,178.718,5.982,149.452
C04930=1146.799,-105.278,-43.786,178.720,5.983,149.451
C04931=1146.794,-105.029,-43.795,178.722,5.984,149.451
C04932=1146.788,-104.779,-43.805,178.724,5.984,149.450
C04933=1146.783,-104.529,-43.814,178.727,5.984,149.449
C04934=1146.778,-104.279,-43.823,178.728,5.984,149.449
C04935=1146.773,-104.029,-43.831,178.730,5.985,149.448
C04936=1146.767,-103.780,-43.840,178.733,5.985,149.448
C04937=1146.761,-103.530,-43.849,178.734,5.985,149.447
C04938=1146.756,-103.280,-43.858,178.736,5.986,149.447
C04939=1146.750,-103.008,-43.869,178.739,5.987,149.446
C04940=1146.744,-102.736,-43.878,178.741,5.987,149.446
C04941=1146.739,-102.464,-43.888,178.743,5.987,149.445
C04942=1146.733,-102.192,-43.899,178.746,5.988,149.445
C04943=1146.728,-101.942,-43.908,178.748,5.988,149.444
C04944=1146.722,-101.693,-43.917,178.749,5.988,149.444
C04945=1146.717,-101.443,-43.925,178.752,5.989,149.443
C04946=1146.711,-101.193,-43.934,178.754,5.989,149.442
C04947=1146.706,-100.943,-43.944,178.756,5.989,149.442
C04948=1146.701,-100.693,-43.953,178.758,5.990,149.441
C04949=1146.696,-100.444,-43.962,178.760,5.990,149.441
C04950=1146.690,-100.194,-43.971,178.762,5.991,149.440
C04951=1146.684,-99.944,-43.981,178.764,5.991,149.440
C04952=1146.679,-99.694,-43.990,178.766,5.991,149.439
C04953=1146.674,-99.444,-43.999,178.768,5.992,149.439
C04954=1146.669,-99.194,-44.009,178.770,5.992,149.438
C04955=1146.663,-98.944,-44.018,178.773,5.992,149.438
C04956=1146.658,-98.695,-44.027,178.775,5.993,149.437
C04957=1146.653,-98.445,-44.037,178.776,5.993,149.437
C04958=1146.647,-98.195,-44.046,178.779,5.994,149.436
C04959=1146.642,-97.945,-44.055,178.780,5.994,149.436
C04960=1146.636,-97.695,-44.064,178.783,5.994,149.435
C04961=1146.631,-97.446,-44.074,178.785,5.995,149.434
C04962=1146.626,-97.196,-44.083,178.787,5.995,149.434
C04963=1146.620,-96.946,-44.092,178.789,5.996,149.433
C04964=1146.615,-96.696,-44.101,178.791,5.996,149.433
C04965=1146.610,-96.447,-44.111,178.793,5.996,149.432
C04966=1146.604,-96.197,-44.120,178.795,5.997,149.432
C04967=1146.599,-95.947,-44.129,178.797,5.997,149.431
C04968=1146.594,-95.698,-44.139,178.799,5.997,149.431
C04969=1146.589,-95.447,-44.148,178.801,5.998,149.430
C04970=1146.583,-95.198,-44.157,178.803,5.998,149.430
C04971=1146.578,-94.948,-44.167,178.806,5.999,149.429
C04972=1146.573,-94.698,-44.176,178.808,5.999,149.429
C04973=1146.567,-94.448,-44.185,178.809,5.999,149.428
C04974=1146.562,-94.199,-44.195,178.812,6.000,149.427
C04975=1146.557,-93.949,-44.204,178.814,6.000,149.427
C04976=1146.551,-93.699,-44.214,178.816,6.000,149.427
C04977=1146.546,-93.450,-44.223,178.818,6.001,149.426
C04978=1146.541,-93.200,-44.232,178.820,6.002,149.426
C04979=1146.535,-92.950,-44.242,178.822,6.001,149.425
C04980=1146.530,-92.700,-44.251,178.824,6.002,149.424
C04981=1146.524,-92.451,-44.261,178.827,6.003,149.424
C04982=1146.519,-92.201,-44.270,178.828,6.003,149.423
C04983=1146.513,-91.951,-44.280,178.831,6.003,149.423
C04984=1146.508,-91.702,-44.289,178.833,6.004,149.422
C04985=1146.503,-91.451,-44.299,178.835,6.004,149.422
C04986=1146.498,-91.202,-44.309,178.837,6.005,149.421
C04987=1146.493,-90.952,-44.317,178.840,6.005,149.420
C04988=1146.487,-90.703,-44.328,178.841,6.005,149.420
C04989=1146.482,-90.453,-44.337,178.843,6.006,149.420
C04990=1146.476,-90.203,-44.347,178.846,6.007,149.419
C04991=1146.471,-89.954,-44.356,178.847,6.007,149.419
C04992=1146.466,-89.703,-44.365,178.850,6.007,149.418
C04993=1146.461,-89.453,-44.375,178.852,6.008,149.417
C04994=1146.455,-89.203,-44.385,178.854,6.008,149.417
C04995=1146.450,-88.954,-44.394,178.856,6.009,149.416
C04996=1146.444,-88.704,-44.404,178.858,6.009,149.416
C04997=1146.439,-88.455,-44.413,178.860,6.009,149.415
C04998=1146.434,-88.205,-44.424,178.862,6.010,149.415
C04999=1146.429,-87.955,-44.432,178.864,6.010,149.414
C05000=1146.423,-87.706,-44.443,178.867,6.010,149.414
C05001=1146.418,-87.456,-44.452,178.869,6.011,149.413
C05002=1146.413,-87.206,-44.462,178.871,6.012,149.413
C05003=1146.408,-86.956,-44.471,178.873,6.011,149.412
C05004=1146.402,-86.706,-44.481,178.875,6.012,149.411
C05005=1146.396,-86.456,-44.491,178.877,6.013,149.411
C05006=1146.391,-86.207,-44.500,178.879,6.013,149.410
C05007=1146.386,-85.957,-44.511,178.881,6.013,149.410
C05008=1146.381,-85.707,-44.519,178.884,6.014,149.409
C05009=1146.375,-85.458,-44.530,178.886,6.014,149.409
C05010=1146.370,-85.207,-44.539,178.888,6.014,149.408
C05011=1146.365,-84.958,-44.549,178.890,6.015,149.408
C05012=1146.360,-84.709,-44.559,178.893,6.016,149.407
C05013=1146.354,-84.458,-44.568,178.894,6.016,149.407
C05014=1146.348,-84.209,-44.578,178.896,6.016,149.406
C05015=1146.344,-83.960,-44.588,178.899,6.017,149.405
C05016=1146.338,-83.709,-44.598,178.901,6.017,149.405
C05017=1146.333,-83.460,-44.608,178.903,6.017,149.404
C05018=1146.327,-83.209,-44.617,178.905,6.018,149.404
C05019=1146.322,-82.960,-44.627,178.908,6.019,149.403
C05020=1146.317,-82.711,-44.637,178.909,6.019,149.403
C05021=1146.311,-82.461,-44.647,178.911,6.019,149.402
C05022=1146.306,-82.210,-44.657,178.914,6.020,149.402
C05023=1146.301,-81.961,-44.667,178.916,6.020,149.401
C05024=1146.296,-81.711,-44.677,178.918,6.020,149.401
C05025=1146.290,-81.462,-44.686,178.920,6.021,149.400
C05026=1146.285,-81.212,-44.696,178.922,6.021,149.399
C05027=1146.280,-80.962,-44.706,178.924,6.022,149.399
C05028=1146.275,-80.712,-44.715,178.927,6.022,149.398
C05029=1146.269,-80.462,-44.725,178.929,6.023,149.398
C05030=1146.264,-80.213,-44.736,178.931,6.023,149.397
C05031=1146.259,-79.964,-44.745,178.933,6.023,149.397
C05032=1146.253,-79.713,-44.755,178.935,6.024,149.396
C05033=1146.248,-79.463,-44.765,178.937,6.025,149.396
C05034=1146.242,-79.214,-44.776,178.939,6.025,149.395
C05035=1146.237,-78.964,-44.785,178.942,6.025,149.395
C05036=1146.232,-78.714,-44.796,178.944,6.026,149.394
C05037=1146.226,-78.464,-44.805,178.946,6.026,149.393
C05038=1146.222,-78.215,-44.815,178.948,6.026,149.393
C05039=1146.216,-77.965,-44.825,178.950,6.027,149.392
C05040=1146.210,-77.716,-44.835,178.952,6.028,149.392
C05041=1146.205,-77.465,-44.846,178.955,6.028,149.391
C05042=1146.200,-77.216,-44.855,178.957,6.028,149.391
C05043=1146.194,-76.944,-44.866,178.959,6.029,149.390
C05044=1146.188,-76.673,-44.877,178.962,6.029,149.390
C05045=1146.183,-76.402,-44.888,178.964,6.030,149.389
C05046=1146.177,-76.130,-44.899,178.966,6.031,149.388
C05047=1146.171,-75.880,-44.909,178.968,6.031,149.388
C05048=1146.166,-75.631,-44.919,178.971,6.031,149.387
C05049=1146.160,-75.381,-44.929,178.973,6.032,149.387
C05050=1146.156,-75.131,-44.939,178.975,6.032,149.386
C05051=1146.150,-74.882,-44.949,178.977,6.032,149.386
C05052=1146.145,-74.632,-44.960,178.979,6.033,149.385
C05053=1146.140,-74.382,-44.970,178.982,6.034,149.385
C05054=1146.134,-74.132,-44.980,178.984,6.034,149.384
C05055=1146.129,-73.883,-44.989,178.986,6.034,149.383
C05056=1146.123,-73.633,-45.000,178.988,6.035,149.383
C05057=1146.118,-73.383,-45.010,178.990,6.035,149.382
C05058=1146.113,-73.133,-45.020,178.993,6.036,149.382
C05059=1146.107,-72.884,-45.031,178.994,6.036,149.381
C05060=1146.102,-72.633,-45.041,178.997,6.037,149.381
C05061=1146.097,-72.384,-45.051,178.999,6.037,149.380
C05062=1146.092,-72.135,-45.061,179.002,6.038,149.380
C05063=1146.087,-71.884,-45.072,179.003,6.038,149.379
C05064=1146.081,-71.635,-45.082,179.005,6.039,149.379
C05065=1146.076,-71.385,-45.092,179.008,6.039,149.378
C05066=1146.071,-71.135,-45.103,179.010,6.040,149.377
C05067=1146.065,-70.886,-45.113,179.012,6.040,149.377
C05068=1146.060,-70.636,-45.122,179.014,6.040,149.376
C05069=1146.055,-70.386,-45.133,179.017,6.041,149.376
C05070=1146.050,-70.137,-45.143,179.019,6.042,149.375
C05071=1146.044,-69.887,-45.153,179.021,6.041,149.375
C05072=1146.039,-69.637,-45.164,179.023,6.042,149.374
C05073=1146.033,-69.387,-45.174,179.025,6.043,149.374
C05074=1146.028,-69.138,-45.184,179.028,6.043,149.373
C05075=1146.023,-68.887,-45.195,179.030,6.044,149.372
C05076=1146.017,-68.638,-45.205,179.032,6.044,149.372
C05077=1146.012,-68.389,-45.215,179.034,6.045,149.371
C05078=1146.008,-68.139,-45.226,179.037,6.045,149.371
C05079=1146.002,-67.889,-45.236,179.039,6.046,149.370
C05080=1145.997,-67.639,-45.247,179.040,6.046,149.370
C05081=1145.991,-67.390,-45.257,179.043,6.046,149.369
C05082=1145.986,-67.140,-45.267,179.045,6.047,149.369
C05083=1145.981,-66.890,-45.278,179.047,6.048,149.368
C05084=1145.975,-66.640,-45.288,179.050,6.048,149.367
C05085=1145.970,-66.390,-45.299,179.052,6.048,149.367
C05086=1145.965,-66.141,-45.309,179.054,6.049,149.366
C05087=1145.959,-65.892,-45.320,179.057,6.049,149.366
C05088=1145.954,-65.641,-45.330,179.059,6.050,149.365
C05089=1145.949,-65.392,-45.340,179.061,6.051,149.365
C05090=1145.944,-65.142,-45.351,179.063,6.050,149.364
C05091=1145.938,-64.892,-45.361,179.065,6.051,149.364
C05092=1145.933,-64.643,-45.372,179.067,6.052,149.363
C05093=1145.928,-64.393,-45.383,179.070,6.052,149.362
C05094=1145.922,-64.143,-45.393,179.072,6.053,149.362
C05095=1145.917,-63.893,-45.404,179.074,6.053,149.361
C05096=1145.912,-63.644,-45.414,179.077,6.053,149.361
C05097=1145.907,-63.394,-45.425,179.079,6.054,149.360
C05098=1145.901,-63.144,-45.435,179.081,6.055,149.360
C05099=1145.896,-62.894,-45.446,179.084,6.055,149.359
C05100=1145.891,-62.645,-45.456,179.085,6.055,149.359
C05101=1145.885,-62.396,-45.467,179.087,6.056,149.358
C05102=1145.880,-62.145,-45.478,179.090,6.056,149.357
C05103=1145.875,-61.896,-45.488,179.092,6.057,149.357
C05104=1145.870,-61.646,-45.498,179.094,6.058,149.356
C05105=1145.865,-61.397,-45.509,179.096,6.058,149.356
C05106=1145.860,-61.146,-45.520,179.099,6.058,149.355
C05107=1145.854,-60.897,-45.530,179.101,6.059,149.355
C05108=1145.849,-60.647,-45.541,179.104,6.060,149.354
C05109=1145.844,-60.398,-45.552,179.106,6.060,149.354
C05110=1145.838,-60.147,-45.563,179.108,6.061,149.353
C05111=1145.833,-59.898,-45.574,179.110,6.061,149.352
C05112=1145.828,-59.648,-45.584,179.112,6.061,149.352
C05113=1145.822,-59.398,-45.594,179.114,6.062,149.351
C05114=1145.817,-59.149,-45.606,179.117,6.063,149.351
C05115=1145.812,-58.899,-45.616,179.119,6.063,149.350
C05116=1145.807,-58.649,-45.626,179.121,6.064,149.350
C05117=1145.801,-58.400,-45.637,179.123,6.064,149.349
C05118=1145.796,-58.150,-45.648,179.126,6.065,149.349
C05119=1145.790,-57.900,-45.659,179.128,6.065,149.348
C05120=1145.785,-57.650,-45.670,179.131,6.066,149.347
C05121=1145.780,-57.401,-45.680,179.133,6.067,149.347
C05122=1145.775,-57.151,-45.692,179.135,6.067,149.346
C05123=1145.770,-56.901,-45.702,179.137,6.067,149.346
C05124=1145.765,-56.652,-45.713,179.139,6.068,149.345
C05125=1145.760,-56.402,-45.724,179.142,6.068,149.345
C05126=1145.754,-56.152,-45.734,179.144,6.069,149.344
C05127=1145.749,-55.902,-45.746,179.146,6.070,149.344
C05128=1145.743,-55.653,-45.756,179.149,6.070,149.343
C05129=1145.739,-55.403,-45.767,179.150,6.070,149.342
C05130=1145.733,-55.154,-45.777,179.153,6.071,149.342
C05131=1145.728,-54.904,-45.789,179.155,6.071,149.341
C05132=1145.723,-54.653,-45.800,179.158,6.072,149.341
C05133=1145.717,-54.405,-45.811,179.160,6.072,149.340
C05134=1145.712,-54.154,-45.821,179.162,6.073,149.340
C05135=1145.707,-53.905,-45.832,179.165,6.074,149.339
C05136=1145.702,-53.655,-45.843,179.167,6.074,149.338
C05137=1145.697,-53.405,-45.855,179.169,6.074,149.338
C05138=1145.691,-53.156,-45.865,179.171,6.075,149.337
C05139=1145.686,-52.906,-45.876,179.174,6.075,149.337
C05140=1145.681,-52.656,-45.886,179.176,6.076,149.336
C05141=1145.675,-52.407,-45.898,179.178,6.077,149.336
C05142=1145.670,-52.156,-45.909,179.181,6.077,149.335
C05143=1145.665,-51.907,-45.920,179.182,6.077,149.335
C05144=1145.660,-51.658,-45.931,179.184,6.078,149.334
C05145=1145.654,-51.408,-45.942,179.187,6.079,149.333
C05146=1145.649,-51.158,-45.953,179.189,6.079,149.333
C05147=1145.644,-50.887,-45.966,179.192,6.080,149.332
C05148=1145.637,-50.617,-45.977,179.194,6.081,149.332
C05149=1145.632,-50.346,-45.989,179.197,6.081,149.331
C05150=1145.627,-50.075,-46.001,179.199,6.082,149.331
C05151=1145.621,-49.826,-46.012,179.202,6.082,149.330
C05152=1145.616,-49.576,-46.023,179.204,6.083,149.329
C05153=1145.611,-49.327,-46.034,179.207,6.083,149.329
C05154=1145.605,-49.076,-46.045,179.209,6.084,149.328
C05155=1145.600,-48.827,-46.057,179.211,6.085,149.328
C05156=1145.595,-48.578,-46.068,179.213,6.084,149.327
C05157=1145.589,-48.327,-46.079,179.215,6.085,149.326
C05158=1145.584,-48.078,-46.090,179.217,6.086,149.326
C05159=1145.579,-47.829,-46.101,179.220,6.086,149.325
C05160=1145.573,-47.578,-46.112,179.222,6.087,149.325
C05161=1145.569,-47.329,-46.124,179.225,6.088,149.324
C05162=1145.563,-47.080,-46.134,179.227,6.088,149.324
C05163=1145.558,-46.829,-46.146,179.229,6.089,149.323
C05164=1145.553,-46.579,-46.157,179.232,6.090,149.322
C05165=1145.548,-46.331,-46.168,179.234,6.090,149.322
C05166=1145.542,-46.081,-46.180,179.236,6.090,149.322
C05167=1145.537,-45.830,-46.190,179.238,6.091,149.321
C05168=1145.532,-45.580,-46.202,179.241,6.091,149.320
C05169=1145.527,-45.332,-46.213,179.243,6.092,149.320
C05170=1145.521,-45.082,-46.225,179.245,6.093,149.319
C05171=1145.516,-44.831,-46.236,179.248,6.093,149.319
C05172=1145.511,-44.582,-46.247,179.250,6.094,149.318
C05173=1145.505,-44.332,-46.258,179.253,6.095,149.318
C05174=1145.501,-44.083,-46.270,179.255,6.095,149.317
C05175=1145.495,-43.833,-46.282,179.257,6.096,149.316
C05176=1145.490,-43.583,-46.292,179.259,6.096,149.316
C05177=1145.484,-43.333,-46.304,179.262,6.096,149.315
C05178=1145.480,-43.084,-46.315,179.264,6.097,149.315
C05179=1145.475,-42.834,-46.326,179.266,6.098,149.314
C05180=1145.469,-42.585,-46.338,179.269,6.098,149.314
C05181=1145.464,-42.335,-46.349,179.271,6.099,149.313
C05182=1145.459,-42.085,-46.361,179.274,6.099,149.312
C05183=1145.454,-41.835,-46.372,179.276,6.100,149.312
C05184=1145.448,-41.586,-46.383,179.278,6.101,149.311
C05185=1145.443,-41.336,-46.394,179.281,6.101,149.311
C05186=1145.438,-41.086,-46.406,179.283,6.102,149.310
C05187=1145.433,-40.837,-46.417,179.285,6.103,149.310
C05188=1145.427,-40.587,-46.429,179.288,6.103,149.309
C05189=1145.422,-40.338,-46.440,179.289,6.103,149.309
C05190=1145.417,-40.088,-46.452,179.292,6.104,149.308
C05191=1145.412,-39.838,-46.463,179.294,6.104,149.307
C05192=1145.406,-39.589,-46.475,179.296,6.105,149.307
C05193=1145.401,-39.339,-46.487,179.299,6.106,149.306
C05194=1145.396,-39.089,-46.497,179.301,6.106,149.306
C05195=1145.390,-38.839,-46.509,179.304,6.107,149.305
C05196=1145.385,-38.589,-46.521,179.306,6.108,149.305
C05197=1145.379,-38.340,-46.532,179.308,6.108,149.304
C05198=1145.375,-38.090,-46.543,179.311,6.109,149.303
C05199=1145.369,-37.840,-46.555,179.313,6.110,149.303
C05200=1145.364,-37.591,-46.567,179.316,6.110,149.302
C05201=1145.359,-37.341,-46.579,179.318,6.111,149.302
C05202=1145.354,-37.091,-46.590,179.320,6.112,149.301
C05203=1145.348,-36.842,-46.601,179.323,6.112,149.301
C05204=1145.343,-36.592,-46.613,179.325,6.113,149.300
C05205=1145.338,-36.343,-46.626,179.328,6.113,149.299
C05206=1145.333,-36.093,-46.637,179.330,6.114,149.299
C05207=1145.328,-35.843,-46.649,179.332,6.115,149.298
C05208=1145.323,-35.594,-46.660,179.334,6.114,149.298
C05209=1145.317,-35.344,-46.672,179.336,6.115,149.297
C05210=1145.312,-35.094,-46.684,179.339,6.116,149.297
C05211=1145.307,-34.845,-46.695,179.341,6.116,149.296
C05212=1145.301,-34.595,-46.707,179.343,6.117,149.296
C05213=1145.296,-34.345,-46.719,179.346,6.118,149.295
C05214=1145.291,-34.095,-46.730,179.348,6.118,149.294
C05215=1145.286,-33.845,-46.742,179.350,6.119,149.294
C05216=1145.280,-33.596,-46.753,179.353,6.120,149.293
C05217=1145.275,-33.347,-46.765,179.355,6.120,149.293
C05218=1145.270,-33.097,-46.777,179.358,6.121,149.292
C05219=1145.265,-32.847,-46.789,179.360,6.122,149.292
C05220=1145.260,-32.598,-46.800,179.362,6.122,149.291
C05221=1145.255,-32.348,-46.812,179.365,6.123,149.290
C05222=1145.249,-32.098,-46.824,179.367,6.124,149.290
C05223=1145.245,-31.849,-46.836,179.370,6.124,149.289
C05224=1145.239,-31.599,-46.848,179.372,6.125,149.289
C05225=1145.234,-31.349,-46.860,179.374,6.125,149.288
C05226=1145.228,-31.100,-46.872,179.377,6.126,149.288
C05227=1145.223,-30.850,-46.883,179.379,6.127,149.287
C05228=1145.218,-30.601,-46.895,179.381,6.127,149.286
C05229=1145.213,-30.351,-46.907,179.384,6.128,149.286
C05230=1145.207,-30.101,-46.919,179.386,6.128,149.285
C05231=1145.202,-29.851,-46.931,179.388,6.129,149.285
C05232=1145.197,-29.602,-46.943,179.391,6.130,149.284
C05233=1145.192,-29.352,-46.955,179.393,6.130,149.284
C05234=1145.186,-29.102,-46.967,179.396,6.131,149.283
C05235=1145.182,-28.852,-46.978,179.398,6.132,149.282
C05236=1145.177,-28.603,-46.991,179.400,6.132,149.282
C05237=1145.171,-28.353,-47.003,179.403,6.133,149.282
C05238=1145.166,-28.103,-47.015,179.405,6.134,149.281
C05239=1145.161,-27.854,-47.027,179.407,6.134,149.280
C05240=1145.156,-27.604,-47.038,179.410,6.135,149.280
C05241=1145.151,-27.354,-47.050,179.412,6.136,149.279
C05242=1145.145,-27.105,-47.063,179.414,6.136,149.279
C05243=1145.140,-26.855,-47.075,179.417,6.137,149.278
C05244=1145.135,-26.605,-47.087,179.419,6.138,149.278
C05245=1145.130,-26.356,-47.099,179.422,6.138,149.277
C05246=1145.125,-26.106,-47.111,179.424,6.139,149.276
C05247=1145.119,-25.856,-47.122,179.426,6.140,149.276
C05248=1145.114,-25.607,-47.135,179.429,6.140,149.275
C05249=1145.109,-25.357,-47.147,179.431,6.141,149.275
C05250=1145.104,-25.108,-47.160,179.434,6.141,149.274
C05251=1145.098,-24.838,-47.172,179.436,6.142,149.274
C05252=1145.092,-24.568,-47.185,179.439,6.143,149.273
C05253=1145.087,-24.297,-47.198,179.441,6.144,149.272
C05254=1145.082,-24.028,-47.211,179.444,6.144,149.272
C05255=1145.076,-23.778,-47.223,179.447,6.145,149.271
C05256=1145.071,-23.528,-47.235,179.449,6.146,149.270
C05257=1145.066,-23.279,-47.248,179.451,6.146,149.270
C05258=1145.060,-23.029,-47.260,179.454,6.147,149.269
C05259=1145.055,-22.780,-47.272,179.456,6.148,149.269
C05260=1145.050,-22.529,-47.285,179.459,6.148,149.268
C05261=1145.045,-22.280,-47.297,179.461,6.149,149.268
C05262=1145.040,-22.030,-47.309,179.463,6.150,149.267
C05263=1145.034,-21.781,-47.322,179.466,6.150,149.267
C05264=1145.029,-21.531,-47.333,179.468,6.151,149.266
C05265=1145.024,-21.281,-47.346,179.470,6.151,149.265
C05266=1145.018,-21.031,-47.358,179.473,6.152,149.265
C05267=1145.013,-20.782,-47.371,179.475,6.153,149.264
C05268=1145.008,-20.532,-47.382,179.478,6.153,149.264
C05269=1145.003,-20.283,-47.395,179.480,6.154,149.263
C05270=1144.998,-20.034,-47.407,179.483,6.155,149.263
C05271=1144.993,-19.784,-47.419,179.485,6.156,149.262
C05272=1144.988,-19.535,-47.432,179.488,6.156,149.261
C05273=1144.982,-19.285,-47.443,179.490,6.157,149.261
C05274=1144.978,-19.035,-47.456,179.492,6.158,149.260
C05275=1144.972,-18.785,-47.470,179.495,6.158,149.260
C05276=1144.967,-18.535,-47.481,179.497,6.159,149.259
C05277=1144.961,-18.286,-47.494,179.500,6.160,149.259
C05278=1144.956,-18.036,-47.506,179.502,6.160,149.258
C05279=1144.951,-17.787,-47.519,179.504,6.161,149.258
C05280=1144.946,-17.537,-47.531,179.507,6.162,149.257
C05281=1144.940,-17.287,-47.543,179.509,6.162,149.256
C05282=1144.936,-17.037,-47.556,179.512,6.163,149.256
C05283=1144.931,-16.788,-47.569,179.514,6.164,149.255
C05284=1144.925,-16.538,-47.580,179.516,6.164,149.255
C05285=1144.920,-16.289,-47.593,179.519,6.166,149.254
C05286=1144.915,-16.039,-47.606,179.521,6.167,149.254
C05287=1144.910,-15.789,-47.618,179.524,6.167,149.253
C05288=1144.905,-15.540,-47.630,179.526,6.168,149.253
C05289=1144.900,-15.290,-47.643,179.529,6.168,149.252
C05290=1144.895,-15.041,-47.656,179.531,6.169,149.251
C05291=1144.889,-14.791,-47.668,179.533,6.170,149.251
C05292=1144.884,-14.541,-47.681,179.536,6.170,149.250
C05293=1144.878,-14.292,-47.693,179.538,6.171,149.250
C05294=1144.874,-14.042,-47.706,179.541,6.171,149.249
C05295=1144.868,-13.792,-47.718,179.543,6.172,149.249
C05296=1144.863,-13.543,-47.731,179.546,6.173,149.248
C05297=1144.858,-13.293,-47.743,179.548,6.174,149.247
C05298=1144.853,-13.044,-47.756,179.550,6.175,149.247
C05299=1144.848,-12.795,-47.769,179.553,6.175,149.246
C05300=1144.842,-12.544,-47.782,179.555,6.176,149.246
C05301=1144.837,-12.294,-47.794,179.558,6.177,149.245
C05302=1144.832,-12.045,-47.807,179.560,6.177,149.245
C05303=1144.827,-11.796,-47.819,179.563,6.178,149.244
C05304=1144.823,-11.546,-47.832,179.565,6.179,149.243
C05305=1144.817,-11.296,-47.845,179.567,6.180,149.243
C05306=1144.811,-11.046,-47.857,179.570,6.180,149.242
C05307=1144.806,-10.797,-47.870,179.573,6.182,149.242
C05308=1144.802,-10.547,-47.883,179.575,6.182,149.241
C05309=1144.796,-10.298,-47.896,179.577,6.183,149.241
C05310=1144.791,-10.048,-47.908,179.580,6.184,149.240
C05311=1144.785,-9.799,-47.921,179.582,6.184,149.240
C05312=1144.781,-9.549,-47.934,179.584,6.185,149.239
C05313=1144.776,-9.299,-47.947,179.587,6.185,149.238
C05314=1144.771,-9.050,-47.960,179.589,6.186,149.238
C05315=1144.765,-8.800,-47.973,179.592,6.186,149.237
C05316=1144.760,-8.550,-47.986,179.595,6.188,149.237
C05317=1144.755,-8.301,-47.998,179.597,6.189,149.236
C05318=1144.750,-8.051,-48.010,179.600,6.189,149.236
C05319=1144.745,-7.801,-48.023,179.602,6.190,149.235
C05320=1144.739,-7.551,-48.036,179.604,6.190,149.234
C05321=1144.734,-7.302,-48.049,179.607,6.191,149.234
C05322=1144.729,-7.053,-48.062,179.609,6.192,149.233
C05323=1144.724,-6.802,-48.075,179.612,6.193,149.233
C05324=1144.719,-6.553,-48.088,179.614,6.194,149.232
C05325=1144.714,-6.304,-48.100,179.617,6.195,149.232
C05326=1144.708,-6.053,-48.114,179.619,6.195,149.231
C05327=1144.704,-5.805,-48.127,179.622,6.196,149.230
C05328=1144.698,-5.555,-48.140,179.624,6.197,149.230
C05329=1144.693,-5.305,-48.153,179.626,6.197,149.230
C05330=1144.688,-5.056,-48.166,179.629,6.199,149.229
C05331=1144.683,-4.806,-48.179,179.631,6.199,149.228
C05332=1144.678,-4.556,-48.192,179.634,6.200,149.228
C05333=1144.673,-4.307,-48.205,179.636,6.201,149.227
C05334=1144.667,-4.058,-48.217,179.639,6.201,149.227
C05335=1144.662,-3.807,-48.231,179.641,6.202,149.226
C05336=1144.657,-3.558,-48.243,179.643,6.203,149.226
C05337=1144.652,-3.309,-48.256,179.647,6.204,149.225
C05338=1144.647,-3.059,-48.270,179.649,6.205,149.224
C05339=1144.642,-2.810,-48.283,179.651,6.205,149.224
C05340=1144.637,-2.560,-48.296,179.654,6.206,149.223
C05341=1144.631,-2.310,-48.309,179.656,6.206,149.223
C05342=1144.626,-2.061,-48.322,179.658,6.207,149.222
C05343=1144.620,-1.811,-48.335,179.661,6.209,149.222
C05344=1144.616,-1.561,-48.348,179.664,6.209,149.221
C05345=1144.610,-1.312,-48.362,179.666,6.210,149.221
C05346=1144.606,-1.062,-48.375,179.669,6.211,149.220
C05347=1144.601,-0.813,-48.387,179.671,6.211,149.219
C05348=1144.595,-0.563,-48.401,179.673,6.212,149.219
C05349=1144.591,-0.314,-48.414,179.676,6.213,149.218
C05350=1144.585,-0.064,-48.427,179.678,6.214,149.218
C05351=1144.580,0.186,-48.440,179.681,6.215,149.217
C05352=1144.574,0.436,-48.454,179.683,6.215,149.217
C05353=1144.570,0.684,-48.467,179.686,6.216,149.216
C05354=1144.564,0.935,-48.480,179.688,6.217,149.215
C05355=1144.559,1.204,-48.494,179.691,6.218,149.215
C05356=1144.553,1.473,-48.509,179.694,6.219,149.214
C05357=1144.548,1.743,-48.523,179.697,6.220,149.214
C05358=1144.543,2.012,-48.537,179.699,6.221,149.213
C05359=1144.537,2.262,-48.551,179.702,6.221,149.212
C05360=1144.532,2.512,-48.564,179.704,6.222,149.212
C05361=1144.527,2.761,-48.578,179.706,6.222,149.211
C05362=1144.522,3.011,-48.590,179.709,6.224,149.211
C05363=1144.517,3.261,-48.604,179.712,6.224,149.210
C05364=1144.511,3.510,-48.618,179.714,6.225,149.210
C05365=1144.506,3.760,-48.631,179.716,6.226,149.209
C05366=1144.501,4.009,-48.644,179.719,6.226,149.209
C05367=1144.496,4.259,-48.657,179.722,6.228,149.208
C05368=1144.491,4.508,-48.671,179.724,6.229,149.207
C05369=1144.486,4.758,-48.684,179.727,6.229,149.207
C05370=1144.480,5.007,-48.698,179.729,6.230,149.206
C05371=1144.476,5.257,-48.710,179.732,6.231,149.206
C05372=1144.470,5.506,-48.724,179.734,6.232,149.205
C05373=1144.465,5.757,-48.738,179.737,6.233,149.205
C05374=1144.460,6.005,-48.751,179.739,6.233,149.204
C05375=1144.455,6.256,-48.765,179.742,6.234,149.203
C05376=1144.450,6.504,-48.778,179.744,6.236,149.203
C05377=1144.445,6.755,-48.792,179.747,6.236,149.203
C05378=1144.439,7.004,-48.806,179.749,6.237,149.202
C05379=1144.435,7.254,-48.819,179.751,6.238,149.201
C05380=1144.430,7.504,-48.833,179.754,6.238,149.201
C05381=1144.424,7.753,-48.846,179.757,6.240,149.200
C05382=1144.420,8.003,-48.860,179.759,6.240,149.200
C05383=1144.414,8.252,-48.873,179.762,6.241,149.199
C05384=1144.409,8.502,-48.887,179.764,6.242,149.199
C05385=1144.404,8.751,-48.900,179.767,6.243,149.198
C05386=1144.399,9.001,-48.914,179.769,6.244,149.197
C05387=1144.393,9.251,-48.927,179.772,6.244,149.197
C05388=1144.389,9.500,-48.941,179.774,6.245,149.196
C05389=1144.384,9.750,-48.955,179.777,6.247,149.196
C05390=1144.378,9.999,-48.968,179.779,6.247,149.195
C05391=1144.374,10.249,-48.982,179.782,6.248,149.195
C05392=1144.368,10.498,-48.995,179.784,6.248,149.194
C05393=1144.363,10.748,-49.010,179.787,6.250,149.194
C05394=1144.357,10.998,-49.023,179.790,6.250,149.193
C05395=1144.353,11.247,-49.036,179.792,6.251,149.192
C05396=1144.348,11.497,-49.051,179.794,6.252,149.192
C05397=1144.342,11.746,-49.064,179.797,6.253,149.191
C05398=1144.337,11.996,-49.078,179.799,6.254,149.191
C05399=1144.332,12.245,-49.092,179.802,6.254,149.190
C05400=1144.327,12.495,-49.105,179.804,6.255,149.190
C05401=1144.322,12.745,-49.119,179.807,6.257,149.189
C05402=1144.317,12.994,-49.133,179.810,6.257,149.189
C05403=1144.312,13.244,-49.146,179.812,6.258,149.188
C05404=1144.307,13.494,-49.161,179.815,6.259,149.187
C05405=1144.302,13.743,-49.174,179.817,6.260,149.187
C05406=1144.297,13.992,-49.189,179.820,6.261,149.186
C05407=1144.291,14.242,-49.202,179.822,6.261,149.186
C05408=1144.287,14.491,-49.216,179.824,6.262,149.185
C05409=1144.282,14.741,-49.230,179.828,6.264,149.185
C05410=1144.276,14.990,-49.244,179.830,6.264,149.184
C05411=1144.271,15.240,-49.257,179.832,6.265,149.183
C05412=1144.266,15.490,-49.272,179.835,6.266,149.183
C05413=1144.260,15.739,-49.286,179.837,6.267,149.183
C05414=1144.256,15.988,-49.299,179.840,6.268,149.182
C05415=1144.251,16.238,-49.313,179.842,6.269,149.181
C05416=1144.245,16.488,-49.327,179.845,6.270,149.181
C05417=1144.240,16.738,-49.341,179.848,6.271,149.180
C05418=1144.235,16.987,-49.355,179.850,6.271,149.180
C05419=1144.230,17.237,-49.370,179.853,6.273,149.179
C05420=1144.225,17.486,-49.383,179.855,6.273,149.179
C05421=1144.221,17.735,-49.397,179.858,6.274,149.178
C05422=1144.215,17.986,-49.411,179.860,6.275,149.178
C05423=1144.210,18.235,-49.425,179.863,6.276,149.177
C05424=1144.205,18.484,-49.439,179.865,6.277,149.176
C05425=1144.200,18.734,-49.453,179.868,6.278,149.176
C05426=1144.194,18.983,-49.467,179.871,6.279,149.175
C05427=1144.189,19.233,-49.481,179.873,6.280,149.175
C05428=1144.184,19.483,-49.496,179.876,6.280,149.174
C05429=1144.179,19.732,-49.510,179.878,6.282,149.174
C05430=1144.174,19.981,-49.524,179.881,6.283,149.173
C05431=1144.169,20.231,-49.538,179.883,6.283,149.173
C05432=1144.164,20.481,-49.552,179.885,6.284,149.172
C05433=1144.159,20.730,-49.567,179.889,6.285,149.171
C05434=1144.153,20.979,-49.581,179.891,6.286,149.171
C05435=1144.148,21.229,-49.595,179.893,6.286,149.170
C05436=1144.144,21.479,-49.609,179.896,6.288,149.170
C05437=1144.139,21.729,-49.623,179.898,6.289,149.169
C05438=1144.134,21.978,-49.638,179.901,6.289,149.169
C05439=1144.128,22.227,-49.652,179.904,6.291,149.168
C05440=1144.123,22.477,-49.666,179.906,6.291,149.168
C05441=1144.118,22.727,-49.680,179.909,6.292,149.167
C05442=1144.113,22.976,-49.694,179.911,6.294,149.167
C05443=1144.108,23.225,-49.708,179.914,6.294,149.166
C05444=1144.103,23.475,-49.723,179.916,6.295,149.165
C05445=1144.098,23.725,-49.737,179.919,6.296,149.165
C05446=1144.093,23.975,-49.751,179.922,6.297,149.164
C05447=1144.088,24.224,-49.765,179.924,6.298,149.164
C05448=1144.083,24.474,-49.780,179.927,6.299,149.163
C05449=1144.077,24.723,-49.794,179.929,6.300,149.163
C05450=1144.072,24.973,-49.808,179.932,6.300,149.162
C05451=1144.068,25.222,-49.823,179.935,6.302,149.162
C05452=1144.063,25.471,-49.837,179.937,6.303,149.161
C05453=1144.058,25.721,-49.851,179.939,6.303,149.160
C05454=1144.052,25.970,-49.865,179.942,6.305,149.160
C05455=1144.047,26.220,-49.880,179.945,6.305,149.159
C05456=1144.042,26.470,-49.894,179.947,6.306,149.159
C05457=1144.037,26.719,-49.909,179.950,6.308,149.158
C05458=1144.032,26.969,-49.924,179.952,6.308,149.158
C05459=1144.027,27.238,-49.939,179.955,6.310,149.157
C05460=1144.021,27.507,-49.954,179.958,6.310,149.157
C05461=1144.016,27.776,-49.971,179.961,6.312,149.156
C05462=1144.010,28.044,-49.986,179.963,6.312,149.156
C05463=1144.005,28.294,-50.000,179.967,6.314,149.155
C05464=1144.000,28.544,-50.015,179.969,6.315,149.154
C05465=1143.995,28.793,-50.029,179.971,6.315,149.154
C05466=1143.990,29.043,-50.045,179.974,6.317,149.153
C05467=1143.985,29.292,-50.059,179.976,6.317,149.153
C05468=1143.980,29.542,-50.073,179.979,6.319,149.152
C05469=1143.975,29.792,-50.087,179.982,6.320,149.152
C05470=1143.970,30.041,-50.102,179.984,6.320,149.151
C05471=1143.964,30.291,-50.117,179.987,6.322,149.151
C05472=1143.959,30.540,-50.131,179.989,6.322,149.150
C05473=1143.954,30.789,-50.146,179.992,6.323,149.149
C05474=1143.949,31.039,-50.160,179.995,6.325,149.149
C05475=1143.944,31.289,-50.175,179.997,6.325,149.148
C05476=1143.939,31.538,-50.190,-180.000,6.327,149.148
C05477=1143.934,31.788,-50.205,-179.998,6.327,149.147
C05478=1143.929,32.037,-50.220,-179.996,6.328,149.147
C05479=1143.924,32.287,-50.234,-179.992,6.330,149.146
C05480=1143.919,32.536,-50.249,-179.990,6.330,149.146
C05481=1143.914,32.785,-50.264,-179.987,6.332,149.145
C05482=1143.909,33.035,-50.278,-179.985,6.332,149.145
C05483=1143.904,33.285,-50.294,-179.983,6.333,149.144
C05484=1143.899,33.534,-50.308,-179.979,6.335,149.144
C05485=1143.894,33.783,-50.323,-179.977,6.335,149.143
C05486=1143.888,34.033,-50.338,-179.974,6.337,149.142
C05487=1143.883,34.283,-50.352,-179.972,6.337,149.142
C05488=1143.879,34.532,-50.367,-179.970,6.338,149.141
C05489=1143.873,34.782,-50.382,-179.966,6.340,149.141
C05490=1143.868,35.031,-50.397,-179.964,6.340,149.140
C05491=1143.863,35.281,-50.411,-179.961,6.342,149.140
C05492=1143.858,35.530,-50.427,-179.959,6.342,149.139
C05493=1143.853,35.780,-50.441,-179.957,6.343,149.139
C05494=1143.848,36.029,-50.456,-179.953,6.345,149.138
C05495=1143.843,36.279,-50.472,-179.951,6.345,149.138
C05496=1143.838,36.528,-50.486,-179.949,6.347,149.137
C05497=1143.833,36.777,-50.501,-179.946,6.348,149.137
